		(*BALANCE*)
		(*************************************************************************************************)
		bI_EnableBalanceLink                                            := TRUE;
		fI_CorrectionValue                                              := 1.00;
		iI_RefreshRate                                                  := 2000;   (*ms*)
		FOR iL_Counter := 1 TO iCIk_NB_INKSTORAGE_TANK DO
			sAdsIkInkStorageTank[iL_Counter].sI_EnableBalance.bI_Command  := TRUE;

			sAdsIkInkStorageTank[iL_Counter].sI_InkDensitySet.fI_Val      := 1.07;
			sAdsIkInkStorageTank[iL_Counter].sI_CorrectionValue.fI_Val    := 1.00;
			sAdsIkInkStorageTank[iL_Counter].fO_StorageTankSize           := 25.0;   (*l*)

			sAdsIkInkStorageTank[iL_Counter].sI_WarningLevelSet.fI_Val    := 4.0;
			sAdsIkInkStorageTank[iL_Counter].sI_ErrorlevelSet.fI_Val      := 3.0;
			sAdsIkInkStorageTank[iL_Counter].sI_MaintenanceTimeout.lI_Val := 5000;

      (*Varnish parameter*)
      sAdsIkInkStorageTank[iL_Counter].sI_InkParameter.aWaveform           := 'waveform.wav';
      sAdsIkInkStorageTank[iL_Counter].sI_InkParameter.sTemperature.fI_Val := 35.0;
      sAdsIkInkStorageTank[iL_Counter].sI_InkParameter.sMeniscus.fI_Val    := -24.5;
      sAdsIkInkStorageTank[iL_Counter].sI_InkParameter.sDensity.fI_Val     := 1.0;
      sAdsIkInkStorageTank[iL_Counter].sI_InkParameter.sViscosity.fI_Val   := 100.0;
		END_FOR

		FOR iL_Counter := 1 TO iCIk_NB_INKBALANCE DO
      fL_BalanceOffset[iL_Counter]                                  := 0;

			sAdsIkInkStorageTank[iL_Counter].aI_CalibrateFrameText1       := 'aaaaaaaa';
			sAdsIkInkStorageTank[iL_Counter].aI_CalibrateFrameText2       := 'bbbbbbbb';
		END_FOR;
		sAdsIkInkStorageTank[1].aI_CalibrateFrameText1                  := '4D5A2406';
		sAdsIkInkStorageTank[1].aI_CalibrateFrameText2                  := '399128E6';
		sAdsIkInkStorageTank[2].aI_CalibrateFrameText1                  := '4D5426F9';
		sAdsIkInkStorageTank[2].aI_CalibrateFrameText2                  := '3991CD5A';
		sAdsIkInkStorageTank[3].aI_CalibrateFrameText1                  := 'aaaaaaaa';
		sAdsIkInkStorageTank[3].aI_CalibrateFrameText2                  := 'bbbbbbbb';

    (*Recipe: load and write*)
    IF pFbRecipeMngr <> 0 THEN
      pFbRecipeMngr^.mWriteRecipe('');
      PRG_MACHINE.bI_RecipeValuesLoadedInk := TRUE;
    END_IF

  ELSE

    sR_RemVar_I.aL_Pattern := sR_RemVar_I.aL_Pattern;  (*TODO remove dummy code*)

    (*DEGASSING*)
    (*************************************************************************************************)
    sAdsIkDgas[1].bI_Enable             := sR_RemVar_I.lR_DgasEnable;
    sAdsIkDgas[1].sI_PressSet.fI_Val    := (sR_RemVar_I.fR_DgasPressStpt * sC_Config_I.fL_DGAS1_CONV_ADS_TO_LCL);

    bIDp_EnableMainDgasValve            := sR_RemVar_I.lR_DgasEnableMainValve;
    sC_Config_I.lL_DGAS_TIME_ERROR      := sR_RemVar_I.lR_DgasTimeError;


    (*MENISCUS*)
    (*************************************************************************************************)
    FOR iL_Counter := 1 TO iCIk_NB_MENC DO
      sAdsIkMenc[iL_Counter].bI_Enable                         := sR_RemVar_I.lR_MencEnable   [iL_Counter];
      sAdsIkMenc[iL_Counter].sI_PressSet.fI_Val                := sR_RemVar_I.fR_MencPressStpt[iL_Counter];
    END_FOR;

    sC_Config_I.wL_MENC_TIME_ERROR                             := sR_RemVar_I.wR_MencTimeError;
    sC_Config_I.wL_SUB_MENC_TIME_ERROR                         := sR_RemVar_I.wR_SubMencTimeError;


    (*SUB MENISCUS*)
    (*************************************************************************************************)
    (*Sub meniscus starts behind the meniscus*)
    FOR iL_Counter := 1 TO iCIk_NB_SUB_MENC DO
      sAdsIkMenc[iCIk_NB_MENC + iL_Counter].bI_Enable          := sR_RemVar_I.lR_SubMencEnable        [iL_Counter];
      sAdsIkMenc[iCIk_NB_MENC + iL_Counter].sI_PressSet.fI_Val := sR_RemVar_I.fR_SubMencPressStpt     [iL_Counter];
    END_FOR;


    (*INK*)
    (*************************************************************************************************)
    (*varnish*)
    FOR iL_Counter := 1 TO iCIk_NB_HEADERTANK DO
      sAdsIkHeaderTank[iL_Counter].sI_StoragetankAssignment.lI_Val    := sR_RemVar_I.lR_StoragetankAssignment[iL_Counter];
      sAdsIkHeaderTank[iL_Counter].sO_ActStoragetankAssignment.lI_Val := sR_RemVar_I.lR_ActStoragetankAssignment[iL_Counter];
      
      sAdsIkHeaderTank[iL_Counter].bI_EnableFillInk       := sR_RemVar_I.bI_EnableFillInk[iL_Counter];
      sAdsIkHeaderTank[iL_Counter].bI_FillModeAuto        := sR_RemVar_I.bI_FillModeAuto[iL_Counter];
      sAdsIkHeaderTank[iL_Counter].bI_EnableUnFillInk     := sR_RemVar_I.bI_EnableUnFillInk[iL_Counter];
      sAdsIkHeaderTank[iL_Counter].bI_UnFillModeAuto      := sR_RemVar_I.bI_UnFillModeAuto[iL_Counter];

      sAdsIkInkPump[iL_Counter].sI_InkPumpSpeedSet.lI_Val := WORD_TO_DINT(sR_RemVar_I.wR_StptSpeedFillInkPumpVarnishPercent[iL_Counter]);

      fb_Headertank[iL_Counter].StateHeadertank           := sR_RemVar_I.eR_StateHeadertank[iL_Counter];
    END_FOR

		wIDp_MinSpeedFillInkPumpVarnish								:= sR_RemVar_I.wR_MinSpeedFillInkPumpVarnish;
		wIDp_MaxSpeedFillInkPumpVarnish								:= sR_RemVar_I.wR_MaxSpeedFillInkPumpVarnish;
		wIDP_AnalogMinDigitVarnish 										:= sR_RemVar_I.wR_AnalogMinDigitVarnish;
		wIDP_AnalogMaxDigitVarnish 										:= sR_RemVar_I.wR_AnalogMaxDigitVarnish;
		wIDp_PumpTimeOffDelayVarnish									:= sR_RemVar_I.wR_PumpTimeOffDelayVarnish;

    lL_TimeReturnFlow                             := sR_RemVar_I.lR_TimeReturnFlow;
    lL_TimeBlowOut                                := sR_RemVar_I.lR_TimeBlowOut;
    lL_TimeEmptyCleaner                           := sR_RemVar_I.lR_TimeEmptyCleaner;
    lL_TimeWarnExchange                           := sR_RemVar_I.lR_TimeWarnExchange;

    sC_Config_I.wC_INKPUMP_MAX_TIME               := sR_RemVar_I.wR_InkPumpMaxTime;
    sC_Config_I.wC_CLEANERPUMP_MAX_TIME           := sR_RemVar_I.wR_CleanerPumpMaxTime;

    
    (*TEMP*)
    (*************************************************************************************************)
    FOR iL_Counter :=1 TO iCIk_NB_TEMP_CONTR DO
      sAdsIkHeater[iL_Counter].bI_EnableHeater     := sR_RemVar_I.bI_EnableHeater  [iL_Counter];
      sAdsIkHeater[iL_Counter].sI_HeaterSet.fI_Val := sR_RemVar_I.sI_HeaterSetPoint[iL_Counter];
    END_FOR


    (*PURGE*)
    (*************************************************************************************************)
    FOR iL_Counter := 1 TO iCIk_NB_PURGE_CONTR DO
      sAdsIkPurgeController[iL_Counter].bI_Enable         := sR_RemVar_I.bR_PurgeControllerEnable[iL_Counter];
    END_FOR;

    FOR iL_Counter := 1 TO iCIk_NB_PURGE_GROUP DO
      sAdsIkPurgeGroup[iL_Counter].bI_EnablePurge         := sR_RemVar_I.bR_PurgeGroupEnable       [iL_Counter];
      sAdsIkPurgeGroup[iL_Counter].bI_EnableThroughNozzle := sR_RemVar_I.bR_PurgeGroupThroughNozzle[iL_Counter];
      sAdsIkPurgeGroup[iL_Counter].bI_EnableFlush         := sR_RemVar_I.bR_PurgeGroupFlush        [iL_Counter];
    END_FOR;


		(*BALANCE*)
		(*************************************************************************************************)
		bI_EnableBalanceLink    := sR_RemVar_I.bI_EnableBalanceLink;
		fI_CorrectionValue      := sR_RemVar_I.fI_CorrectionValue;
		iI_RefreshRate          := sR_RemVar_I.iI_RefreshRate;
		iI_MaintenanceTimeout   := sR_RemVar_I.iI_MaintenanceTimeout;

		FOR iL_Counter := 1 TO iCIk_NB_INKSTORAGE_TANK DO
			sAdsIkInkStorageTank[iL_Counter].bI_EnableStorageTank        := sR_RemVar_I.bI_EnableStorageTank[iL_Counter];
			sAdsIkInkStorageTank[iL_Counter].lO_InkColorId               := sR_RemVar_I.lO_InkColorId[iL_Counter];
			sAdsIkInkStorageTank[iL_Counter].fO_StorageTankSize          := sR_RemVar_I.fO_StorageTankSize[iL_Counter];
		END_FOR;

		FOR iL_Counter := 1 TO iCIk_NB_INKBALANCE DO
			sAdsIkInkStorageTank[iL_Counter].sI_EnableBalance.bI_Command := sR_RemVar_I.bI_EnableBalance[iL_Counter];
			sAdsIkInkStorageTank[iL_Counter].sI_InkDensitySet.fI_Val     := sR_RemVar_I.sI_InkDensitySet[iL_Counter];
			sAdsIkInkStorageTank[iL_Counter].sI_CorrectionValue.fI_Val   := sR_RemVar_I.sI_CorrectionValue[iL_Counter];
			sAdsIkInkStorageTank[iL_Counter].sI_WarningLevelSet.fI_Val   := sR_RemVar_I.sI_WarningLevelSet[iL_Counter];
			sAdsIkInkStorageTank[iL_Counter].sI_ErrorlevelSet.fI_Val     := sR_RemVar_I.sI_ErrorlevelSet[iL_Counter];

      (*Varnish parameter*)
      sAdsIkInkStorageTank[iL_Counter].sI_InkParameter.iScannerId          := sR_RemVar_I.lR_VarParamScannerId[iL_Counter];
      sAdsIkInkStorageTank[iL_Counter].sI_InkParameter.iIndex              := sR_RemVar_I.iR_VarParamIndex[iL_Counter];
      sAdsIkInkStorageTank[iL_Counter].sI_InkParameter.sTemperature.fI_Val := sR_RemVar_I.fR_VarParamTemp[iL_Counter];
      sAdsIkInkStorageTank[iL_Counter].sI_InkParameter.sMeniscus.fI_Val    := sR_RemVar_I.fR_VarParamMenc[iL_Counter];
      sAdsIkInkStorageTank[iL_Counter].sI_InkParameter.aWaveform           := sR_RemVar_I.aR_VarParamWaveform[iL_Counter];
      sAdsIkInkStorageTank[iL_Counter].sI_InkParameter.iTimer              := sR_RemVar_I.iR_VarParamTimer[iL_Counter];
      sAdsIkInkStorageTank[iL_Counter].sI_InkParameter.sDensity.fI_Val     := sR_RemVar_I.fR_VarParamDensity[iL_Counter];
      sAdsIkInkStorageTank[iL_Counter].sI_InkParameter.sViscosity.fI_Val   := sR_RemVar_I.fR_VarParamViscosity[iL_Counter];
      sAdsIkInkStorageTank[iL_Counter].sI_InkParameter.iColorId            := sR_RemVar_I.iR_VarParamColorId[iL_Counter];
      FOR iL_Counter2 := 1 TO 10 DO
        sAdsIkInkStorageTank[iL_Counter].sI_InkParameter.bCompatibility[iL_Counter2] := sR_RemVar_I.bR_VarParamCompatibility[iL_Counter, iL_Counter2];
      END_FOR;

			sAdsIkInkStorageTank[iL_Counter].aI_CalibrateFrameText1      := sR_RemVar_I.aI_CalibrateFrameText1[iL_Counter];
			sAdsIkInkStorageTank[iL_Counter].aI_CalibrateFrameText2      := sR_RemVar_I.aI_CalibrateFrameText2[iL_Counter];

      fL_BalanceOffset[iL_Counter] := sR_RemVar_I.fR_BalanceOffset[iL_Counter];
		END_FOR;

  END_IF


  bL_RemVar_Init := FALSE;



(*************************************************************************************************)
(********************************* WRITING REMANENT VARIABLES ************************************)
(*************************************************************************************************)
ELSE

(*GENERAL*)
(*************************************************************************************************)
  sR_RemVar_I.aL_Pattern := 16#ABCD;

(*DEGASSING*)
(*************************************************************************************************)
  sR_RemVar_I.lR_DgasEnable           := sAdsIkDgas[1].bI_Enable;
  sR_RemVar_I.fR_DgasPressStpt        := sAdsIkDgas[1].sI_PressSet.fI_Val;

  sR_RemVar_I.lR_DgasEnableMainValve  := bIDp_EnableMainDgasValve;
  sR_RemVar_I.lR_DgasTimeError        := sC_Config_I.lL_DGAS_TIME_ERROR;

(*MENISCUS*)
(*************************************************************************************************)
  FOR iL_Counter := 1 TO iCIk_NB_MENC DO
    sR_RemVar_I.fR_MencPressStpt[iL_Counter]      := sAdsIkMenc[iL_Counter].sI_PressSet.fI_Val;
    sR_RemVar_I.lR_MencEnable   [iL_Counter]      := sAdsIkMenc[iL_Counter].bI_Enable;
  END_FOR;

  sR_RemVar_I.wR_MencTimeError                    := sC_Config_I.wL_MENC_TIME_ERROR;
  sR_RemVar_I.wR_SubMencTimeError                 := sC_Config_I.wL_SUB_MENC_TIME_ERROR;

(*SUB MENISCUS*)
(*************************************************************************************************)
  (*Sub meniscus starts behind the meniscus*)
  FOR iL_Counter := 1 TO iCIk_NB_SUB_MENC DO
    sR_RemVar_I.fR_SubMencPressStpt     [iL_Counter] := sAdsIkMenc[iCIk_NB_MENC + iL_Counter].sI_PressSet.fI_Val;
    sR_RemVar_I.lR_SubMencEnable        [iL_Counter] := sAdsIkMenc[iCIk_NB_MENC + iL_Counter].bI_Enable;
  END_FOR;

(*PURGE - GLOBAL*)
(*************************************************************************************************)
  FOR iL_Counter := 1 TO iCIk_NB_PURGE_CONTR DO
    sR_RemVar_I.bR_PurgeControllerEnable  [iL_Counter] := sAdsIkPurgeController[iL_Counter].bI_Enable;
  END_FOR;

  FOR iL_Counter := 1 TO iCIk_NB_PURGE_GROUP DO
    sR_RemVar_I.bR_PurgeGroupEnable       [iL_Counter] := sAdsIkPurgeGroup[iL_Counter].bI_EnablePurge;
    sR_RemVar_I.bR_PurgeGroupThroughNozzle[iL_Counter] := sAdsIkPurgeGroup[iL_Counter].bI_EnableThroughNozzle;
    sR_RemVar_I.bR_PurgeGroupFlush        [iL_Counter] := sAdsIkPurgeGroup[iL_Counter].bI_EnableFlush;
  END_FOR;


(*INK*)
(*************************************************************************************************)
  (*varnish*)
  FOR iL_Counter:= 1 TO iCIk_NB_HEADERTANK DO
    sR_RemVar_I.lR_StoragetankAssignment   [iL_Counter]           := sAdsIkHeaderTank[iL_Counter].sI_StoragetankAssignment.lI_Val;
    sR_RemVar_I.lR_ActStoragetankAssignment[iL_Counter]           := sAdsIkHeaderTank[iL_Counter].sO_ActStoragetankAssignment.lI_Val;
      
    sR_RemVar_I.bI_EnableFillInk  [iL_Counter]                    := sAdsIkHeaderTank[iL_Counter].bI_EnableFillInk;
    sR_RemVar_I.bI_FillModeAuto   [iL_Counter]                    := sAdsIkHeaderTank[iL_Counter].bI_FillModeAuto;
    sR_RemVar_I.bI_EnableUnFillInk[iL_Counter]                    := sAdsIkHeaderTank[iL_Counter].bI_EnableUnFillInk;
    sR_RemVar_I.bI_UnFillModeAuto [iL_Counter]                    := sAdsIkHeaderTank[iL_Counter].bI_UnFillModeAuto;

    sR_RemVar_I.wR_StptSpeedFillInkPumpVarnishPercent[iL_Counter] := DINT_TO_WORD(sAdsIkInkPump[iL_Counter].sI_InkPumpSpeedSet.lI_Val);
    
    sR_RemVar_I.eR_StateHeadertank[iL_Counter]                    := fb_Headertank[iL_Counter].StateHeadertank;
  END_FOR

	sR_RemVar_I.wR_MinSpeedFillInkPumpVarnish 				:= wIDp_MinSpeedFillInkPumpVarnish;
	sR_RemVar_I.wR_MaxSpeedFillInkPumpVarnish					:= wIDp_MaxSpeedFillInkPumpVarnish;
	sR_RemVar_I.wR_AnalogMinDigitVarnish 							:= wIDP_AnalogMinDigitVarnish;
	sR_RemVar_I.wR_AnalogMaxDigitVarnish 							:= wIDP_AnalogMaxDigitVarnish;
	sR_RemVar_I.wR_PumpTimeOffDelayVarnish 						:= wIDp_PumpTimeOffDelayVarnish;

  sR_RemVar_I.lR_TimeReturnFlow                     := lL_TimeReturnFlow;
  sR_RemVar_I.lR_TimeBlowOut                        := lL_TimeBlowOut;
  sR_RemVar_I.lR_TimeEmptyCleaner                   := lL_TimeEmptyCleaner;
  sR_RemVar_I.lR_TimeWarnExchange                   := lL_TimeWarnExchange;

  sR_RemVar_I.wR_InkPumpMaxTime                     := sC_Config_I.wC_INKPUMP_MAX_TIME;
  sR_RemVar_I.wR_CleanerPumpMaxTime                 := sC_Config_I.wC_CLEANERPUMP_MAX_TIME;


(*RAMPE*)
(*************************************************************************************************)


(*TEMP*)
(*************************************************************************************************)
  FOR iL_Counter := 1 TO iCIk_NB_TEMP_CONTR DO
    sR_RemVar_I.bI_EnableHeater  [iL_Counter] := sAdsIkHeater[iL_Counter].bI_EnableHeater;
    sR_RemVar_I.sI_HeaterSetPoint[iL_Counter] := sAdsIkHeater[iL_Counter].sI_HeaterSet.fI_Val;
  END_FOR

  
(*INKSTORAGE_TANK*)
(*************************************************************************************************)
  FOR iL_Counter := 1 TO iCIk_NB_INKSTORAGE_TANK DO
    sR_RemVar_I.bI_EnableStorageTank[iL_Counter] := sAdsIkInkStorageTank[iL_Counter].bI_EnableStorageTank;
    sR_RemVar_I.lO_InkColorId[iL_Counter]        := sAdsIkInkStorageTank[iL_Counter].lO_InkColorId;
    sR_RemVar_I.fO_StorageTankSize[iL_Counter]   := sAdsIkInkStorageTank[iL_Counter].fO_StorageTankSize;
  END_FOR;

	(*BALANCE*)
	sR_RemVar_I.bI_EnableBalanceLink  := bI_EnableBalanceLink;
	sR_RemVar_I.fI_CorrectionValue    := fI_CorrectionValue;
	sR_RemVar_I.iI_RefreshRate        := iI_RefreshRate;
	sR_RemVar_I.iI_MaintenanceTimeout := iI_MaintenanceTimeout;

  FOR iL_Counter := 1 TO iCIk_NB_INKBALANCE DO
    sR_RemVar_I.bI_EnableBalance    [iL_Counter]   := sAdsIkInkStorageTank[iL_Counter].sI_EnableBalance.bI_Command;
    sR_RemVar_I.sI_InkDensitySet    [iL_Counter]   := sAdsIkInkStorageTank[iL_Counter].sI_InkDensitySet.fI_Val;
    sR_RemVar_I.sI_CorrectionValue  [iL_Counter]   := sAdsIkInkStorageTank[iL_Counter].sI_CorrectionValue.fI_Val;
    sR_RemVar_I.sI_WarningLevelSet  [iL_Counter]   := sAdsIkInkStorageTank[iL_Counter].sI_WarningLevelSet.fI_Val;
    sR_RemVar_I.sI_ErrorlevelSet    [iL_Counter]   := sAdsIkInkStorageTank[iL_Counter].sI_ErrorlevelSet.fI_Val;

    (*Varnish parameter*)
    sR_RemVar_I.lR_VarParamScannerId[iL_Counter]   := sAdsIkInkStorageTank[iL_Counter].sI_InkParameter.iScannerId;
    sR_RemVar_I.iR_VarParamIndex    [iL_Counter]   := sAdsIkInkStorageTank[iL_Counter].sI_InkParameter.iIndex;
    sR_RemVar_I.fR_VarParamTemp     [iL_Counter]   := sAdsIkInkStorageTank[iL_Counter].sI_InkParameter.sTemperature.fI_Val;
    sR_RemVar_I.fR_VarParamMenc     [iL_Counter]   := sAdsIkInkStorageTank[iL_Counter].sI_InkParameter.sMeniscus.fI_Val;
    sR_RemVar_I.aR_VarParamWaveform [iL_Counter]   := sAdsIkInkStorageTank[iL_Counter].sI_InkParameter.aWaveform;
    sR_RemVar_I.iR_VarParamTimer    [iL_Counter]   := sAdsIkInkStorageTank[iL_Counter].sI_InkParameter.iTimer;
    sR_RemVar_I.fR_VarParamDensity  [iL_Counter]   := sAdsIkInkStorageTank[iL_Counter].sI_InkParameter.sDensity.fI_Val;
    sR_RemVar_I.fR_VarParamViscosity[iL_Counter]   := sAdsIkInkStorageTank[iL_Counter].sI_InkParameter.sViscosity.fI_Val;
    sR_RemVar_I.iR_VarParamColorId  [iL_Counter]   := sAdsIkInkStorageTank[iL_Counter].sI_InkParameter.iColorId;
    FOR iL_Counter2 := 1 TO 10 DO
      sR_RemVar_I.bR_VarParamCompatibility[iL_Counter, iL_Counter2] := sAdsIkInkStorageTank[iL_Counter].sI_InkParameter.bCompatibility[iL_Counter2];
    END_FOR;

    sR_RemVar_I.aI_CalibrateFrameText1[iL_Counter] := sAdsIkInkStorageTank[iL_Counter].aI_CalibrateFrameText1;
    sR_RemVar_I.aI_CalibrateFrameText2[iL_Counter] := sAdsIkInkStorageTank[iL_Counter].aI_CalibrateFrameText2;

    sR_RemVar_I.fR_BalanceOffset[iL_Counter] := fL_BalanceOffset[iL_Counter];
  END_FOR;

END_IF;
END_ACTION

ACTION Simulate:
IF bL_SimInputs THEN
  
  FOR iL_CounterDgas := 1 TO iCIk_NB_DGAS DO
    fb_DgasMencContr[iL_CounterDgas].iI_ActValue := LREAL_TO_INT(fb_DgasMencContr[iL_CounterDgas].pSetValue * fb_DgasMencContr[iL_CounterDgas].fR_ConvAdsToLocal);
  
    sAdsIkDgas[iL_CounterDgas].bI_Enable := TRUE;
  END_FOR
  
  FOR iL_CounterMenc := 1 TO iCIk_NB_MENC_STA DO
    fb_MeniscusMencContr[iL_CounterMenc].iI_ActValue := LREAL_TO_INT(fb_MeniscusMencContr[iL_CounterMenc].pSetValue * fb_MeniscusMencContr[iL_CounterMenc].fR_ConvAdsToLocal);
  
    sAdsIkMenc[iL_CounterMenc].bI_Enable := TRUE;
  END_FOR
  
  bIKn_TankCleanerLevelEmpty := TRUE;
  bIKn_TankRefuseLevelFull   := TRUE;
  
  FOR iL_Counter := 1 TO iCIk_NB_TEMP_HYS DO
    fb_TempControllerHys[iL_Counter].iI_ActValue := DINT_TO_INT(fb_TempControllerHys[iL_Counter].pSetValue);
  END_FOR
END_IF

// init any storage tank assignement
FOR iL_Counter := 1 TO iCIk_NB_HEADERTANK DO
  IF sAdsIkHeaderTank[iL_Counter].sI_StoragetankAssignment.lI_Val = 0 THEN
    sAdsIkHeaderTank[iL_Counter].sI_StoragetankAssignment.lI_Val := UDINT_TO_DINT(sL_BLK_INKSTORAGE_TANK[1].iBlk_AdsId);
	END_IF
END_FOR
END_ACTION

ACTION Visu:
(*call visu controls*)
fb_VisuDgasMencController    (sI_Ary_Fb := fb_DgasMencContr    , sI_Ary_Ads := sAdsIkDgas);
fb_VisuMeniscusMencController(sI_Ary_Fb := fb_MeniscusMencContr, sI_Ary_Ads := sAdsIkMenc);
END_ACTION

END_PROGRAM

// ---- POUs/Products/Ink/FB_PurgeControllerSequence.TcPOU
FUNCTION_BLOCK FB_PurgeControllerSequence EXTENDS FB_PurgeController
VAR_INPUT
  iSubMencPos                  : I_AirVolume;
  iSubMencNeg                  : I_AirVolume;
END_VAR

VAR_OUTPUT
  bO_DeactivateLevelControlHT  : BOOL;
  bO_DeactivateSubMencNeg      : BOOL;

  bO_PurgeReleaseValveDelayed  AT %Q* : BOOL;              (*Purge pressure release valve*)
END_VAR

VAR
  _bActivateSequence           : BOOL;

  iL_PurgeStep                 : INT := 0;
  fb_TonSubMencRelease         : TON;
  fb_TonSubMencReleaseDelay    : TON;
  fb_TonSubMencReactivate      : TON;
  fb_RTrigCommand              : R_TRIG;
  fb_SubMencPosRamp            : FB_SPEED_RAMP;
  fb_SubMencNegRamp            : FB_SPEED_RAMP;
END_VAR

VAR PERSISTENT
  tR_ReleaseTime               : TIME := T#3S;
  tR_SubMencReleaseDelay       : TIME := T#1S;
  tR_SubMencReactivateTime     : TIME := T#2S;
  iR_SubMencPosFactor          : INT  := 50;
  iR_SubMencNegFactor          : INT  := 50;
  tR_SubMencPosRampTime        : INT  := 10;
  tR_SubMencNegRampTime        : INT  := 10;
END_VAR

VAR CONSTANT
  iC_StepIdle                  : INT := 0;
  iC_StepMencRelease           : INT := 1;
  iC_StepLevelContr            : INT := 2;
  iC_StepPurge                 : INT := 3;
  iC_StepReactivate1           : INT := 4;
  iC_StepReactivate2           : INT := 5;
END_VAR

(*Delay for one ReleaseValve*)
bO_PurgeReleaseValveDelayed := fbPurgeGroup[1].bO_PurgeReleaseValve;

IF _bActivateSequence THEN
  CASE iL_PurgeStep OF
    iC_StepIdle:  (*Idle, wait for start command*)
      IF     (   _pAdsIf^.sI_ActivatePurge.bI_Command
              OR IbPurgeContrRequestHT
              OR (iMachineInk.pPurgeRequest AND (   _pAdsIf^.sI_ActivatePurge.bO_CommandCanEx
                                                 OR bL_PurgeAuto)))
         AND _pAdsIf^.sI_ActivatePurge.bO_CommandCanEx
      THEN
        _pAdsIf^.sI_ActivatePurge.bO_CommandExec := TRUE;
        _pAdsIf^.sI_ActivatePurge.bI_Command     := FALSE;
  
        fb_TonSubMencRelease(IN := FALSE);
        FOR iL_CounterPurgeGroup := 1 TO iL_RegPurgeGroupItfs DO
          fb_TonSubMencReleaseDelay(IN := FALSE);
        END_FOR
        fb_RTrigCommand(CLK := _pAdsIf^.sI_ActivatePurge.bI_Command);
  
        fb_SubMencPosRamp(bI_EnableRamp := TRUE, bI_StartRamp := FALSE, II_SpeedActPercent := 100);
        fb_SubMencNegRamp(bI_EnableRamp := TRUE, bI_StartRamp := FALSE, II_SpeedActPercent := 100);
  
        iL_PurgeStep := iC_StepMencRelease;
      ELSE
        SUPER^();  
  
        bO_DeactivateLevelControlHT := FALSE;
        bO_DeactivateSubMencNeg     := FALSE;
      END_IF
  
    iC_StepMencRelease:  (*Release sub menc pressure*)
      fb_TonSubMencRelease(IN:= TRUE, PT := tR_ReleaseTime);
  
      FOR iL_CounterPurgeGroup := 1 TO iL_RegPurgeGroupItfs DO
        fb_TonSubMencReleaseDelay(IN := TRUE, PT := tR_SubMencReleaseDelay);
        bO_PurgeReleaseValveDelayed := fb_TonSubMencReleaseDelay.Q;
  
        fbPurgeGroup[iL_CounterPurgeGroup].pEnableValve := TRUE;
      END_FOR
      
      IF fb_TonSubMencRelease.Q THEN
        iL_PurgeStep := iC_StepLevelContr;
      END_IF
    
      (*Abort Purge*)
      fb_RTrigCommand(CLK := _pAdsIf^.sI_ActivatePurge.bI_Command);
      IF fb_RTrigCommand.Q THEN
        fb_TonSubMencReactivate(IN := FALSE);
  
        iL_PurgeStep := iC_StepReactivate1;
      END_IF
    
    iC_StepLevelContr:
      bO_DeactivateLevelControlHT := TRUE;
  
      _pAdsIf^.sI_ActivatePurge.bI_Command := TRUE;
    
      iL_PurgeStep := iC_StepPurge;
    
    iC_StepPurge:
      SUPER^();  
      IF _bBusy THEN
        _pAdsIf^.sI_ActivatePurge.bI_Command := FALSE;
      ELSE
        fb_TonSubMencReactivate(IN := FALSE);
  
        iL_PurgeStep := iC_StepReactivate1;
      END_IF
  
    iC_StepReactivate1:
      fb_TonSubMencReactivate(IN:= TRUE, PT := tR_SubMencReactivateTime);
  
      (*SubMenc must be run up by ramp*)
      fb_SubMencPosRamp( bI_StartRamp         := TRUE
                       , II_XTimeRamp         := tR_SubMencPosRampTime
                       , II_YAnalogMinPercent := iR_SubMencPosFactor
                       , II_YAnalogMaxPercent := 100);
      iSubMencPos.pPressSetFactor := DINT_TO_REAL(fb_SubMencPosRamp.IO_YPercent) / 100;
      
      bO_DeactivateLevelControlHT := FALSE;
      bO_DeactivateSubMencNeg     := TRUE;
  
      _pAdsIf^.sI_ActivatePurge.bO_CommandExec := FALSE;
      _pAdsIf^.sI_ActivatePurge.bI_Command     := FALSE;
  
      FOR iL_CounterPurgeGroup := 1 TO iL_RegPurgeGroupItfs DO
        fbPurgeGroup[iL_CounterPurgeGroup].pEnableValve := FALSE;
      END_FOR
  
      IF fb_TonSubMencReactivate.Q THEN
        iL_PurgeStep := iC_StepReactivate2;
      END_IF
    
    iC_StepReactivate2:
      (*SubMenc must be run up by ramp*)
      fb_SubMencPosRamp( bI_StartRamp         := TRUE
                       , II_XTimeRamp         := tR_SubMencPosRampTime
                       , II_YAnalogMinPercent := iR_SubMencPosFactor
                       , II_YAnalogMaxPercent := 100);
      iSubMencPos.pPressSetFactor := DINT_TO_REAL(fb_SubMencPosRamp.IO_YPercent) / 100;
      fb_SubMencNegRamp( bI_StartRamp         := TRUE
                       , II_XTimeRamp         := tR_SubMencNegRampTime
                       , II_YAnalogMinPercent := iR_SubMencNegFactor
                       , II_YAnalogMaxPercent := 100);
      iSubMencNeg.pPressSetFactor := DINT_TO_REAL(fb_SubMencNegRamp.IO_YPercent) / 100;
  
      bO_DeactivateSubMencNeg := FALSE;
  
      IF fb_SubMencPosRamp.bO_MaxSpeedReached AND fb_SubMencNegRamp.bO_MaxSpeedReached THEN
        iSubMencPos.pPressSetFactor := 1;
        iSubMencNeg.pPressSetFactor := 1;
        
        iL_PurgeStep := iC_StepIdle;
      END_IF
    
  END_CASE
ELSE
  SUPER^();  
END_IF

PROPERTY pActivateSequence : BOOL
SET
_bActivateSequence := pActivateSequence;
END_SET
END_PROPERTY

END_FUNCTION_BLOCK

// ---- POUs/Products/Ink/InkCirculation/FB_InkCirculation.TcPOU
FUNCTION_BLOCK FB_InkCirculation EXTENDS FB_BaseInk IMPLEMENTS I_SleepObserver, I_EmergencyObserver

VAR_INPUT
  InActValue                 AT %I* : INT;                      (*Actual value*)
  IbActValueWcState          AT %I* : BOOL;                     (*EM3701 pressure WcState*)
  IbInkLevelReachedBack      AT %I* : BOOL;                     (*HT back level reached*)

  iPurgeController                  : I_Purge;
  iMencController                   : I_AirVolume;

  IbEnable                          : BOOL;                     (*Enable function*)
  IbAxisMovement                    : BOOL;                     (*Axis movement*)
  IbHeadertankOk                    : BOOL;                     (*Headertank ok*)
  IbPHTempOk                        : BOOL;                     (*Printhead temperature ok*)
END_VAR

VAR_OUTPUT
  ObHtCloseInkConnectionValve       : BOOL;                     (*HT: close ink connection valve front to back*)
  ObHtCloseMencConnectionValve      : BOOL;                     (*HT back: close menc connection valve*)
  ObValveActivation                 : BOOL;                     (*HT: valve activation*)
  ObPumpActivation                  : BOOL;                     (*HT: pump activation*)
END_VAR

VAR
  _sName                            : STRING;                   (*Block name*)

  _bEStop                           : BOOL := FALSE;            (*EStop active*)
  _bSleep                           : BOOL := FALSE;            (*Sleep active*)
  bCheckParameterError01            : BOOL := FALSE;            (*CheckParameter: error 01 reported*)
  bLevelError                       : BOOL := FALSE;            (*HT back level error*)
  bCirculationActive                : BOOL;                     (*Circulation active*)
  bConditionsMet                    : BOOL;                     (*Conditions met*)
  bPumpActivation                   : BOOL;                     (*HT: pump activation*)
  fbTpPumpOn                        : TP;                       (*HT: pump activation on*)
  tPumpOnTime                       : TIME;                     (*HT: pump activation on*)
  fbTpPumpWait                      : TP;                       (*HT: pump activation wait*)
  tPumpWaitTime                     : TIME;                     (*HT: pump activation wait*)
  bResetErrorCounter                : BOOL;                     (*Reset HT back level error counter*)

  fbTonSubMencOK                    : TON;                      (*Sub menc pressure ok*)
  fbTonNoMovement                   : TON;                      (*No axis movement active*)
  fbTonResumeCirculation            : TON;                      (*Resume circulation after level error*)

  fSubMencActValue                  : LREAL;                    (*HT: actual pressure of back side*)
  fSubMencTargetValue               : LREAL;                    (*HT: target pressure of back side*)
END_VAR

VAR PERSISTENT
  tRSubMencOk                       : TIME := T#5S;             (*Supervision time for sub menc ok*)
  tRNoMovement                      : TIME := T#1M;             (*Supervision time axis movement*)
  tRResumeCirculation               : TIME := T#1M;             (*Resume circulation after level error*)
  tRPumpDutyCycleFrequency          : TIME := T#100MS;          (*Frequency for duty cycle of pump*)
  nRPumpDutyCycle                   : UINT := 30;               (*Duty cycle of pump*)

  fRConvAdsToLocal                  : LREAL := 10.0;            (*Factor to convert from ADS to local*)
  fRSubMencDeltaP                   : LREAL := -2.5;            (*HT: delta pressure of sub menc on back side*)
  fRSubMencHysteresisP              : LREAL :=  0.5;            (*HT: hysteresis pressure*)
  fRSubMencCorrectionP              : LREAL :=  0.0;            (*HT: correction pressure*)

  nRErrorCounter                    : UINT := 0;                (*HT back level error counter*)
END_VAR

(*--- check parameter -------------------*)
IF NOT mCheckParameter() THEN RETURN; END_IF

(*HT back error*)
IF bCirculationActive AND IbInkLevelReachedBack THEN
  bLevelError    := TRUE;
  nRErrorCounter := nRErrorCounter + 1;
END_IF
fbTonResumeCirculation(IN := bLevelError, PT := tRResumeCirculation);
IF fbTonResumeCirculation.Q THEN
  bLevelError    := FALSE;
END_IF
IF bResetErrorCounter THEN
  nRErrorCounter := 0;
END_IF

fbTonSubMencOK (IN := (iMencController.pErrorCode = 0), PT := tRSubMencOk);
fbTonNoMovement(IN := NOT IbAxisMovement, PT := tRNoMovement);

fSubMencActValue    := INT_TO_LREAL(InActValue) / fRConvAdsToLocal;
fSubMencActValue    := fSubMencActValue + fRSubMencCorrectionP;
fSubMencTargetValue := iMencController.pPressure + fRSubMencDeltaP;

bConditionsMet :=     NOT IbActValueWcState
                  AND NOT _bEStop
                  AND NOT _bSleep
                  AND NOT IbInkLevelReachedBack
                  AND NOT bLevelError
                  AND NOT iPurgeController.pPurgeBusy
                  AND fbTonSubMencOK.Q
                  AND fbTonNoMovement.Q
                  AND IbHeadertankOk
                  AND IbPHTempOk
                  AND (fRSubMencDeltaP <> 0);

IF IbEnable AND bConditionsMet THEN
  bCirculationActive           := TRUE;
  ObHtCloseInkConnectionValve  := TRUE;
  ObHtCloseMencConnectionValve := TRUE;
  ObValveActivation            := TRUE;

  IF fSubMencActValue >= (fSubMencTargetValue + fRSubMencHysteresisP) THEN
    bPumpActivation := TRUE;
  END_IF
  IF fSubMencActValue <= (fSubMencTargetValue - fRSubMencHysteresisP) THEN
    bPumpActivation := FALSE;
  END_IF
ELSE  
  bCirculationActive           := FALSE;
  ObHtCloseInkConnectionValve  := FALSE;
  ObHtCloseMencConnectionValve := FALSE;
  ObValveActivation            := FALSE;
  bPumpActivation              := FALSE;
END_IF

(*Pump is activated with a variable duty cycle*)
tPumpOnTime   := DINT_TO_TIME((TIME_TO_DINT(tRPumpDutyCycleFrequency) * nRPumpDutyCycle) / 100);
tPumpWaitTime := DINT_TO_TIME((TIME_TO_DINT(tRPumpDutyCycleFrequency) * (100 - nRPumpDutyCycle)) / 100);
IF bPumpActivation THEN
  IF (nRPumpDutyCycle = 0) THEN
    ObPumpActivation := FALSE;
  ELSIF (nRPumpDutyCycle = 100) THEN
    ObPumpActivation := TRUE;
  ELSE
    fbTpPumpOn  (IN := NOT fbTpPumpWait.Q, PT := tPumpOnTime);
    fbTpPumpWait(IN := NOT fbTpPumpOn.Q  , PT := tPumpWaitTime);
  
    ObPumpActivation := fbTpPumpOn.Q;
  END_IF
ELSE
  fbTpPumpOn  (IN := FALSE);
  fbTpPumpWait(IN := FALSE);

  ObPumpActivation := FALSE;
END_IF

(*
  Check if all necessary variables are properly defined 
  - check if initialized
  - crash prevention!
*)
METHOD PRIVATE mCheckParameter : BOOL
IF (iPurgeController = 0) OR (iMencController = 0) THEN
  IF NOT bCheckParameterError01 THEN
    bCheckParameterError01 := TRUE;
    F_Report_Error(Report_Error_0Pointer);
  END_IF
  RETURN;
END_IF

mCheckParameter := TRUE; // all params ok
END_METHOD

METHOD mEmergencyUpdate
VAR_INPUT
	(*updated estop value TRUE = active*)
	bEStop	: BOOL;
END_VAR
_bEStop := bEStop;
END_METHOD

METHOD mSleepUpdate
VAR_INPUT
	(*updated sleep value TRUE = active*)
	bSleep	: BOOL;
END_VAR
_bSleep := bSleep;
END_METHOD

PROPERTY pName : STRING
SET
_sName := pName;
END_SET
END_PROPERTY

END_FUNCTION_BLOCK

// ---- POUs/Projects/Machine/PRG_MACHINE.TcPOU
PROGRAM PRG_MACHINE
(*************************************************************************************************)
(*  FILENAME:    PRG_MACHINE.EXP                                                                 *)
(*  PROJECT:     CALMAR PUPLC                                                                    *)
(*  COPYRIGHT:   All rights reserved (c) Wifag//Polytype, Fribourg/Switzerland (2016)            *)
(*  ENVIRONMENT: TwinCAT PLC                                                                     *)
(*  VERSION:     <version>                                                                       *)
(*************************************************************************************************)
(*  DESCRIPTION:                                                                   <description> *)
(*    Controls the machine functionalities.                                                      *)
(*     - System command: sleep/wake up, emergency stop, air ok.                                  *)
(*    Messaging: - fb_Msg[1] := `eCMa_EMERGENCY_STOP_ACTIVE`                                     *)
(*               - fb_Msg[2] := `eCMa_MACHINE_DISABLED`                                          *)
(*               - fb_Msg[3] := `eCMa_MACHINE_COMM_ERR`                                          *)
(*               - fb_Msg[4] := `eCMa_SLEEP_MODE_ACTIVE`                                         *)
(*               - fb_Msg[5] := `eCMa_TEMPERATURE_MONITORING`                                    *)
(*               - fb_Msg[6] := `eCMa_STOR_TANKS_DISABLED`                                       *)
(*               - fb_Msg[7] := `eCMa_INK_WC_STATE_ERROR`                                        *)
(*               - fb_Msg[8] := `eCMa_PRINT_WC_STATE_ERROR`                                      *)
(*               - fb_Msg[9] := `eCMa_MACHINE_WC_STATE_ERROR`                                    *)
(*               - fb_Msg[10]:= `eCMa_TCPIP_COMM_ERROR`                                          *)
(*               - fb_Msg[11]:= `eCIk_CLEANER_CONTAINER_LEVEL_EMPTY`                             *)
(*               - fb_Msg[12]:= `eCIk_REFUSE_CONTAINER_LEVEL_FULL`                               *)
(*               - fb_Msg[13]:= `eCMa_AXIS_ERROR_X_PNEUMATIC`                                    *)
(*               - fb_Msg[14]:= `eCMa_WATCH_CIRCUIT_BREAKER`                                     *)
(*               - fb_Msg[15]:= `eCMa_WATCH_FUSE_PH1`                                            *)
(*               - fb_Msg[16]:= `eCMa_WATCH_FUSE_HEATER1`                                        *)
(*               - fb_Msg[17]:= `eCMa_WATCH_CABINET_TEMP`                                        *)
(*               - fb_Msg[18]:= `eCMa_WATCH_SEPARATOR_NIVEAU`                                    *)
(*               - fb_Msg[19]:= `eCMa_AXIS_SAFETY_ACCEPTANCE`                                    *)
(*               - fb_Msg[20]:= `eCMa_DRIFT_CONTR_ERROR`                                         *)
(*               - fb_Msg[21]:= `eCIk_CLEAN_START_MISSING`                                       *)
(*               - fb_Msg[22]:= `eCMa_RECIPE_LOADED`                                             *)
(*               - fb_Msg[23]:= `eCMa_AXIS_ERROR_Z_PNEUMATIC`                                    *)
(*               - fb_Msg[24]:= `eCMa_CLEANER_TANK_INFO`                                         *)
(*               - fb_Msg[25]:= `eCMa_MAX_SPEED_EXCEEDED`                                        *)
(*               - fb_Msg[26]:= `eCMa_IMAGE_DEPTH_INCORRECT`                                     *)
(*               - fb_Msg[27]:= `eCMa_EXHAUST_SYSTEM_WARNING`                                    *)
(*               - fb_Msg[28]:= `eCMa_EXHAUST_SYSTEM_ERROR`                                      *)
(*               - fb_Msg[29]:= `eCMa_EXHAUST_SYSTEM_MALFUNCTION`                                *)
(*               - fb_Msg[30]:= `eCMa_CLEANER_TANK_FILLING`                                      *)
(*               - fb_Msg[31]:= `eCMa_SEPARATOR_LEVEL_REACHED`                                   *)
(*                                                                                </description> *)
(*************************************************************************************************)

VAR_INPUT
  bIKp_CircuitBreakerM1_Ok          AT %I*  : BOOL;   (*monitoring input*)
  bIKp_CircuitBreakerM2_Ok          AT %I*  : BOOL;   (*monitoring input*)
  bIKp_PowerSupply1M1_Ok            AT %I*  : BOOL;   (*monitoring input*)
  bIKp_PowerSupply2M1_Ok            AT %I*  : BOOL;   (*monitoring input*)
  bIKp_PowerSupply3M1_Ok            AT %I*  : BOOL;   (*monitoring input*)
  bIKp_PowerSupply1M2_Ok            AT %I*  : BOOL;   (*monitoring input*)
  bIKp_PowerSupply2M2_Ok            AT %I*  : BOOL;   (*monitoring input*)
  bIKp_PowerSupply3M2_Ok            AT %I*  : BOOL;   (*monitoring input*)
  bIKp_SefetyRelayOk                AT %I*  : ARRAY[1..iCPr_NB_PM] OF BOOL;   (*monitoring input*)
  bIKp_SafetyCoverOK                AT %I*  : ARRAY[1..iCPr_NB_PM] OF BOOL;   (*monitoring input*)
  bIKp_SafetyDoorsOK                AT %I*  : ARRAY[1..iCPr_NB_PM] OF BOOL;   (*monitoring input*)

  bIKp_CabinetTemp_Ok               AT %I*  : BOOL;   (*monitoring input*)
  bIKp_SeparatorNiveau_Ok           AT %I*  : ARRAY[1..iCPr_NB_PM] OF BOOL;   (*-BX66: monitoring input*)
  
  (*Beckhoff EAP interface*)
  InEAP_WatchdogCycleIndex          AT %I*  : INT;    (*Watchdog: check CycleIndex*)
  InEAP_OperatingMode               AT %I*  : BYTE;   (*Operating mode*)
  IbEAP_ShutDownActive              AT %I*  : BOOL;   (*Master is shutting down*)                          (*not used yet*)
  IbEAP_Engaged                     AT %I*  : ARRAY[1..iCPr_NB_PM] OF BOOL;   (*DEM engaged*)
  IbEAP_PrintEnabled                AT %I*  : ARRAY[1..iCPr_NB_PM] OF BOOL;   (*Print enabled*)
  IbEAP_EStop                       AT %I*  : BOOL;   (*Emergency stop*)
  IbEAP_StandbyActive               AT %I*  : BOOL;   (*Standby active*)
  IbEAP_MessageReset                AT %I*  : BOOL;   (*Message reset*)       (*used in PRG_System*)
  IbEAP_PinningClosed               AT %I*  : ARRAY[1..iCPr_NB_PM] OF BOOL;   (*Pinning shutter closed*)
  IbEAP_CleaningStart               AT %I*  : ARRAY[1..iCPr_NB_PM] OF BOOL;   (*Start cleaning*)           (*not used yet*)
  InEAP_SubstrateThickness          AT %I*  : DINT;   (*Substrate thickness [µm]*)
  InEAP_SubstrateWidth              AT %I*  : DINT;   (*Substrate width [µm]*)                             (*not used yet*)
  InEAP_FormatLength                AT %I*  : DINT;   (*Format length [µm]*)
  InEAP_WebStretchFactor            AT %I*  : DINT;   (*Web stretch factor [0/00]*)
  InEAP_LateralRegister             AT %I*  : DINT;   (*Lateral register [µm]*)
  IbEAP_SpliceDetected              AT %I*  : ARRAY[1..iCPr_NB_PM] OF BOOL;   (*Splice detected*)
  InEAP_Module2ToModule3            AT %I*  : DINT;   (*Distance between Module 2 and 3 [µm]*)
  IbEAP_TargetSpeedReached          AT %I*  : BOOL;   (*Target speed reached*)
  InEAP_NeutralFibreFactor          AT %I*  : DINT;   (*Neutral fibre factor [%]*)
  IbEAP_PrintMarksExist             AT %I*  : ARRAY[1..iCPr_NB_PM] OF BOOL;   (*Print marks exist*)
  InEAP_TargetSpeed                 AT %I*  : DINT;   (*Neutral fibre factor [m/min]*)
  IbEAP_PanelLEDs                   AT %I*  : ARRAY[1..nC_MOTRONIC_PANEL_LEDS] OF BOOL;           (*Motronic panel LEDs*)

  (*Interfaces from other PRG*)
  fI_PrintingPosition                       : REAL;   (*Printing position [mm]*)
  bI_RecipeValuesLoadedInk                  : BOOL;
  bI_RecipeValuesLoadedPrint                : BOOL;
  bI_PrintActive                            : BOOL;   (*Printing active*)
  //bI_MachineStopped                         : BOOL;   (*Machine stopped*)
  sI_JobInkConsumption                      : ST_JOB_INK_CONSUMPTION; (*Job ink consumption information*)
  bI_PrintUnitStart                         : BOOL;   (*Printing unit start*)
  bI_PrintUnitStop                          : BOOL;   (*Printing unit stop*)
  lI_PrintedCopies                          : UDINT;  (*Printed copies*)
  bI_VacuumOk                               : BOOL;
  bI_CommandPrintlineExec                   : ARRAY[1..iCPr_NB_PM] OF BOOL;   (*Printline is executing*)

  (*Simulation*)
  bSimulation                               : BOOL;
END_VAR

VAR_OUTPUT
  bOKp_ResetFuse                    AT %Q*  : BOOL;   (*Reset WAGO Epsitron fuse*)
  ObPrinterReady                    AT %Q*  : BOOL;   (*Printer ready*)

  bO_SeparatorPumpDrainage          AT %Q*  : ARRAY[1..iCMa_NB_Cp] OF BOOL;   (* Enable separator pump for tank drainage (-MX196)*)

  bO_InitOk                                 : BOOL := FALSE;  (*Init Ok*)

  bO_WEUReady                               : ARRAY[1..iCPr_NB_PM] OF BOOL;  (*WEU ready*)

  (*Beckhoff EAP interface*)
  OnEAP_OperatingMode               AT %Q*  : BYTE;   (*Operating mode*)
  ObEAP_EngagingAllowed             AT %Q*  : ARRAY[1..iCPr_NB_PM] OF BOOL;   (*DEM engaging allowed*)
  ObEAP_EngagingActive              AT %Q*  : ARRAY[1..iCPr_NB_PM] OF BOOL;   (*DEM engaging active*)
  ObEAP_ShutdownReady               AT %Q*  : BOOL;   (*Shutdown ready*)
  ObEAP_StandbyReady                AT %Q*  : BOOL;   (*Standby ready*)
  ObEAP_PrintPosition               AT %Q*  : ARRAY[1..iCPr_NB_PM] OF BOOL;   (*Printing position*)
  ObEAP_MismatchLength              AT %Q*  : BOOL;   (*Mismatch length*)                               (*not used yet*)
  ObEAP_CleaningAllowed             AT %Q*  : ARRAY[1..iCPr_NB_PM] OF BOOL;   (*Cleaning allowed*)      (*not used yet*)
  ObEAP_CleaningActive              AT %Q*  : ARRAY[1..iCPr_NB_PM] OF BOOL;   (*Cleaning active*)
(*ToDo!!!*)   ObEAP_PrintReady                  AT %Q*  : ARRAY[1..iCPr_NB_PM] OF BOOL;   (*Ready to print*)
  OnEAP_VarnishQuantity             AT %Q*  : ARRAY[1..iCPr_NB_PM] OF DINT;   (*Varnish quantity [g/m^2]*)
  OnEAP_MaxWebSpeed                 AT %Q*  : DINT;   (*Max web speed [m/min]*)
  ObEAP_WarnungActive               AT %Q*  : BOOL;   (*Warning active*)
  ObEAP_ErrorActive                 AT %Q*  : BOOL;   (*Error active*)
  ObEAP_EStop                       AT %Q*  : BOOL;   (*Emergency stop / Fast stop*)
  OnEAP_PrintMarkPosBits            AT %Q*  : ARRAY[1..iCPr_NB_PM] OF WORD;   (*Print mark position (bit coded)*)
                                                                              (*Bit 0: no mark*)
                                                                              (*Bit 1: mark on drive side*)
                                                                              (*Bit 2: mark in center range*)
                                                                              (*Bit 3: mark on control side*)
  OnEAP_MasterSpeed                 AT %Q*  : ARRAY[1..iCPr_NB_PM] OF LREAL;  (*FB_POSITION_MASTER[x].fO_Master_Speed [m/s]*)
  ObPanelLEDs                       AT %Q*  : ARRAY[1..nC_MOTRONIC_PANEL_LEDS] OF BOOL;    (*Motronic panel LEDs*)

  (*Interfaces to other PRG*)
  bO_PrintUnitInPrintPosition               : ARRAY[1..iCPr_NB_PM] OF BOOL;    (*Print unit in print position*)
  bO_PrintUnitHigherWaitPosition            : ARRAY[1..iCPr_NB_PM] OF BOOL;    (*Print unit higher wait position*)
  bO_CleanPumpRequest                       : ARRAY[1..iCMa_NB_Cp] OF BOOL;    (* Request Cleaner Pump on*)
  sO_SystemCmd                              : ST_SYSTEM_CMD;
  bO_TotalWcState                           : BOOL := FALSE;   (*Monitoring: WcStates from all terminals*)
  bO_ErrorMsgActive                         : BOOL;   (*Error message at PUC active*)
  bO_WarningMsgActive                       : BOOL;   (*Warning message at PUC active*)
END_VAR

VAR
  iL_Counter                                : INT;    (*local iteration counter - default*)

  tskL_ActTaskInfo                          : PlcTaskSystemInfo;  (*CycleTime in multiple of 100ns*)
  Fb_GetCurTskIndx                          : GETCURTASKINDEX;
  lL_TaskCycleTime                          : REAL;  (*task cycle time [s]*)

  (* FB to store the generated block ID's *)
  bL_ExecuteBlockIdSave                     : BOOL;
  fb_BlkIdSave                              : FB_BLK_ID_SAVE;

  iL_Sel_BlkType                            : INT  := 1;          (*used for module information visualisation*)

  (*FAF: new cleaning station*)
  fB_Machine                                : FB_MachineState;
  
  fb_CleanProcess                           : ARRAY[1..iCMa_NB_Cp] OF FB_CleaningProcess;
  fb_CleaningCU                             : ARRAY[1..iCMa_NB_Cp] OF FB_CleaningMotorAxisCU;
  fb_CleaningCH                             : ARRAY[1..iCMa_NB_Cp] OF FB_CleaningMotorAxisCH;
  fb_CleaningPU                             : ARRAY[1..iCMa_NB_Cp] OF FB_CleaningMotorAxisPU;
  fb_CleaningValvePump                      : ARRAY[1..iCMa_NB_Cp] OF FB_Cleaning_ValvePump;
  fb_MotionInterlock                        : ARRAY[1..iCMa_NB_Cp] OF FB_MOTION_INTERLOCK;
  bL_RefKnownAll                            : BOOL;
  bL_AllInPosCappingClean                   : BOOL;

  (*Purge from machine*)
  fb_RFTrigPurgeBusy                        : ARRAY[1..iCMa_NB_Cp] OF RF_TRIG;
  fb_RFTrigCleanAfterPurge                  : ARRAY[1..iCMa_NB_Cp] OF RF_TRIG;
  fb_RTrigPurge                             : ARRAY[1..iCMa_NB_Cp] OF R_TRIG;
  fb_TonPurgeRequestTimeout                 : ARRAY[1..iCMa_NB_Cp] OF TON;

  fb_InterfaceMachineInk                    : ARRAY[1..iCPr_NB_PM] OF FB_IMachineInk;
  iMachineInk                               : ARRAY[1..iCPr_NB_PM] OF I_MachineInk;

  fb_MotionInkInterface                     : ARRAY[1..iCPr_NB_PM] OF FB_MOTION_TO_INKSYSTEM_IF;

  //fb_CU_EL7201                              : ARRAY[1..iCMa_NB_Cp] OF FB_EL7201_AXIS_CTRL;
  //fb_CH_EL7201                              : ARRAY[1..iCMa_NB_Cp] OF FB_EL7201_AXIS_CTRL;
  //fb_PU_EL7201                              : ARRAY[1..iCMa_NB_Cp] OF FB_EL7201_001_AXIS_CTRL;
  //lLCU_OffsetEncoder                        : ARRAY[1..iCMa_NB_Cp] OF DINT := [0,0];
  //lLCH_OffsetEncoder                        : ARRAY[1..iCMa_NB_Cp] OF DINT := [0,0];
  //lLPU_OffsetEncoder                        : ARRAY[1..iCMa_NB_Cp] OF DINT := [0,0];
  fb_RFTrigManualMoveCU                     : ARRAY[1..iCMa_NB_Cp] OF RF_TRIG;
  fb_RFTrigManualMoveCH                     : ARRAY[1..iCMa_NB_Cp] OF RF_TRIG;
  fb_RFTrigManualMovePU                     : ARRAY[1..iCMa_NB_Cp] OF RF_TRIG;
  sL_CU_CleanDevStatus                      : ARRAY[1..iCMa_NB_Cp] OF ST_CLEANING_DEV_STATUS;
  sL_CH_CleanDevStatus                      : ARRAY[1..iCMa_NB_Cp] OF ST_CLEANING_DEV_STATUS;
  sL_PU_CleanDevStatus                      : ARRAY[1..iCMa_NB_Cp] OF ST_CLEANING_DEV_STATUS;

  sADS_CleanProcess                         : ARRAY[1..iCMa_NB_Cp] OF ST_ADS_CLEAN_PROCESS;
  sADS_CleanAxis                            : ARRAY[1..iCMa_NB_Ca] OF ST_ADS_CLEAN_AXIS;
  sADS_Machine                              : ARRAY[1..iCMa_NB_Ma] OF ST_ADS_MACHINE;
  sC_Ads_Info                               : ST_ADS_INFO;
  sMappingInfo                              : T_MapInfo;        // Block mapping configuration
  ISystemBase                               : I_SystemBase;     // reference to system base
  pModuleDef                                : POINTER TO FB_ModuleDef;    // Module definition in system
  iSystemCmd                                : I_SystemCmd;                // System Command interface
  iSystemStatus                             : I_SystemStatus;             // System Status interface
  bAllowSleepFromMachine                    : BOOL;                       // enter sleep is allowed from machine
  rfTrig_Estop                              : RF_TRIG;
  
  
  bL_SafetyOk                               : ARRAY[1..iCPr_NB_PM] OF BOOL;
  bL_ResetAxis                              : BOOL;
  bL_MemMachineOn                           : BOOL := FALSE;

  (*Inputs from VISU*)
  (*
  nPrintModuleIdx                           : INT := 1;   (*PrintModule actual selection*)      
  fL_CuCappPurgPosition                     : REAL;  (*CU: capping/purge position [mm]*)
  fL_CuCleanRowPosition1                    : REAL;  (*CU: clean position 1 [mm]*)
  fL_CuCleanRowPosition2                    : REAL;  (*CU: clean position 2 [mm]*)
  fL_CuStopPosition                         : REAL;  (*CU: position ID for the lower limit [mm]*)
  fL_CuPlaceSpeed                           : REAL;  (*CU: speed for placement mouvement [mm/s]*)
  fL_CuWorkSpeed                            : REAL;  (*CU: speed for work mouvement [mm/s]*)
  fL_CuServiceSpeed                         : REAL;  (*CU: speed for maintenance operations [mm/s]*)
  fL_ChPositionP1                           : REAL;  (*CH: position P1 [mm]*)
  fL_ChPositionP2                           : REAL;  (*CH: position P2 [mm]*)
  fL_ChStopPosition                         : REAL;  (*CH: position ID for the lower limit [mm]*)
  fL_ChPlaceSpeed                           : REAL;  (*CH: speed for placement mouvement [mm/s]*)
  fL_ChWorkSpeed                            : REAL;  (*CH: speed for work mouvement [mm/s]*)
  fL_ChServiceSpeed                         : REAL;  (*CH: speed for maintenance operations [mm/s]*)
  fL_PuWaitingPosition                      : REAL;  (*PU: waiting position (Production Mode) [mm]*)
  fL_PuServicePosition                      : REAL;  (*PU: service position (Service Mode) [mm]*)
  fL_PuCleanPosition1                       : REAL;  (*PU: cleaning station moving position (Service Mode) [mm]*)
  fL_PuCleanPosition2                       : REAL;  (*PU: cleaning position (Service Mode) [mm]*)
  fL_PuStopPosition                         : REAL;  (*PU: position ID for the lower limit [mm]*)
  //fL_PuSetPositionValue                     : REAL;  (*PU: set position value [mm]*)
  fL_PuPlaceSpeed                           : REAL;  (*PU: speed for placement mouvement [mm/s]*)
  fL_PuWorkSpeed                            : REAL;  (*PU: speed for work mouvement [mm/s]*)
  fL_PuServiceSpeed                         : REAL;  (*PU: speed for maintenance operations [mm/s]*)
  wIDp_CleanerPumpLeadTime                  : WORD;  (*CH: lead time cleaner pump [ms]*)
  *)
  
  (*Initiation*)
  bL_RemVar_Init                            : BOOL;
  bL_DummyReadInput                         : BOOL;
  iL_DummyReadInput                         : INT;
  lL_DummyReadInput                         : DINT;

  fb_TonCheckMachineCom                     : TON;
  iL_MemWatchdogCycleIndex                  : INT;    (*Watchdog: check CycleIndex*)
  bL_WatchdogError                          : BOOL;

  (*Machine IOs*)
  bL_IO_MachineReady                        : BOOL;
  bL_IO_MachineHoming                       : BOOL;
  bL_IO_Engaged                             : ARRAY[1..iCPr_NB_PM] OF BOOL;
  //bL_IO_EStopOK                             : BOOL;
  bL_IO_StandbyActive                       : BOOL;
  bL_IO_PinningClosed                       : BOOL;
  lL_IO_SubstrateThickness                  : DINT;   (*Substrate thickness [µm]*)
  lL_IO_SubstrateWidth                      : DINT;   (*Substrate width [µm]*)
  lL_IO_FormatLength                        : DINT;   (*Format length [µm]*)
  fb_TonSeparatorLevel                      : ARRAY[1..iCMa_NB_Cp] OF TON;
  bL_SeparatorLevelReached                  : BOOL;

  bL_ProductionMode                         : ARRAY[1..iCPr_NB_PM] OF BOOL;   (*Production mode, not service mode*)

  bL_SleepVisu                              : BOOL;
  bL_WakeUpVisu                             : BOOL;
  fb_RTrigShutdownActive                    : R_TRIG;
  fb_FTrigShutdownActive                    : F_TRIG;
  fb_RTrigOpModeHoming                      : R_TRIG;
  fb_RTrigEngaged                           : ARRAY[1..iCPr_NB_PM] OF R_TRIG;
  fb_FTrigEngaged                           : ARRAY[1..iCPr_NB_PM] OF F_TRIG;
  fb_TonSleepToMachine                      : TON;

  fb_CappingCommandAfterEStop               : FB_CappingCommand;
  fb_CappingCommandAfterError               : ARRAY[1..iCPr_NB_PM] OF FB_CappingCommand;
  fb_CappingCommandAfterEngaged             : ARRAY[1..iCPr_NB_PM] OF FB_CappingCommand;
  fb_CappingCommandAfterShutdown            : ARRAY[1..iCPr_NB_PM] OF FB_CappingCommand;
  fb_CappingCommandAfterCleaning            : ARRAY[1..iCPr_NB_PM] OF FB_CappingCommand;
  _bCappingCommandAfterCleaning             : ARRAY[1..iCPr_NB_PM] OF BOOL;

  fb_TonAxisReady                           : ARRAY[1..iCPr_NB_PM] OF TON;
  fb_TonAxisReadyRelease                    : ARRAY[1..iCPr_NB_PM] OF TON;
  fb_RTrigCleaningFromMachine               : ARRAY[1..iCPr_NB_PM] OF R_TRIG;
  bL_CleaningCommandFromMachine             : ARRAY[1..iCPr_NB_PM] OF BOOL;
	fb_TofCleaningActive                      : ARRAY[1..iCPr_NB_PM] OF TOF;
  
  fb_TofPrintSystemOk                       : TOF;

  sC_Config_M                               : ST_CONFIG_M;

  (*Separator pump for tank drainage*)
  fb_TofSeparatorPumpNiveau                 : ARRAY[1..iCMa_NB_Cp] OF TOF;
  fb_TofSeparatorPumpPurge                  : ARRAY[1..iCMa_NB_Cp] OF TOF;

  bL_ManualVacuumBin                        : ARRAY[1..iCMa_NB_Cp] OF BOOL := [FALSE,FALSE];
  fb_RTrigManualVacuumBin                   : ARRAY[1..iCMa_NB_Cp] OF R_TRIG;
  fb_FTrigManualVacuumBin                   : ARRAY[1..iCMa_NB_Cp] OF F_TRIG;
  fb_RTrigPurgeVacuumBin                    : ARRAY[1..iCMa_NB_Cp] OF R_TRIG;
  fb_FTrigPurgeVacuumBin                    : ARRAY[1..iCMa_NB_Cp] OF F_TRIG;
  fb_FTrigSeparatorNiveau                   : ARRAY[1..iCMa_NB_Cp] OF F_TRIG;

  (*Compare sheet length with Image depth.*)
  lL_SubstrateLenPx                         : DINT;       (*Length of substrate [Px]*)
  lL_ImageDepthPx                           : DINT;       (*Image depth [Px]*)
  lL_ToleranceLenPx                         : DINT := 5;  (*Tolerance for compare sheet length with image depth [Px]*)
  bL_MismatchLength                         : BOOL;       (*Mismatch between length of substrate and image depth*)

  (*Messages*)
  fb_MsgQueueMachine                        : ARRAY [1..iCMa_NB_Ma] OF FB_MSG_QUEUE;
  fb_MachineMsgHandler                      : ARRAY [1..iCMa_NB_Ma] OF FB_MSG_HANDLER;
  sL_MsgConfigMachine                       : ARRAY [1..iCMa_NB_Ma] OF ST_MSG_CONFIG;
  fb_MachineMsg                             : ARRAY [1..iCMa_NB_Ma, 1..iCMa_NB_MSG] OF FB_MESSAGE;

  fb_TpResetFuse                            : TP;

  (*Machine communication NEW*)
  fbMachineComm                             : FB_MachineComm;
  
  (*Epsitron fuse control*)
  fbPowerControl                            : FB_WeuPowerControl;

  (*Exhaust system*)
  fb_ExhaustSystem                          :  ARRAY [1..iCPr_NB_PM] OF FB_ExhaustSystemPrint;
  

(* ADS Mappping *)
(*************************************************************************************************)
  iL_I                                      : INT;                (*instance counter*)
  iL_I2                                     : INT;                (*second instance counter for double loops*)
  sL_pI                                     : POINTER TO ST_MAP_BLK;  (*pointer to module mapping instance*)
  iL_Ctr                                    : INT;                (*counter value*)
  pL_Ctr                                    : POINTER TO INT;      (*pointer to mapping array index*)
  iL_ActElmt                                : INT;                (*actual array element*)
  aL_Name                                   : STRING;              (*Block string creation*)
  iL_NumModules                             : INT;                (*number of different block types*)
  cL_Module                                 : BYTE;                (*this module number*)

  FB_GEN_BLOCK_MAPPING                      : FB_GEN_BLOCK_MAPPING;   (*generation of block mappings in this module*)
  Fb_RegToAry                               : FB_REG_TO_ARY;      (**)

  sL_MOD_MAP                                : ARRAY [1..iCMa_NB_BLOCK_TYPES] OF ST_MAP_MODBLKARY;  (*array conataining all modules with their mapping informations*)
  sL_ModBlkAry                              : ST_MAP_MODBLKARY;

  sL_BLK_MA                                 : ARRAY [1..iCMa_NB_Ma] OF ST_MAP_BLK;      (*Machine*)
  sL_BLK_CP                                 : ARRAY [1..iCMa_NB_Cp] OF ST_MAP_BLK;      (*Cleaning process controller*)
  sL_BLK_AX                                 : ARRAY [1..iCMa_NB_Ca] OF ST_MAP_BLK;      (*array of all cleaning axes*)

  (*Recipe read/write*)
  pFbRecipeMngr                             : POINTER TO FB_RECIPE_READ_WRITE;
  bL_RecipeValuesLoadedMachine              : BOOL;

  (*Simulation variables*)
  bL_SimInputs                              : BOOL := FALSE;
END_VAR

VAR CONSTANT
(*GENERAL*)
(*************************************************************************************************)
  fC_TOLERANCE_PRINT_POSITION               : REAL := 0.001;       (*Tolerance for print position [m]*)

  cC_INIT                                   : BYTE := 16#00;      (*Operating mode: init*)
  cC_INITIALISED                            : BYTE := 16#00;      (*Operating mode: initialised*)
  cC_HOMING                                 : BYTE := 16#01;      (*Operating mode: homing*)
  cC_BASIC_HALT                             : BYTE := 16#02;      (*Operating mode: basic halt*)

  tC_DELAY_CAPPING_COMMAND                  : TIME := T#500MS;    (*Delay for automatic generated capping commands*)
  tC_RELEASE_CAPPING_COMMAND                : TIME := T#2S;       (*Release for automatic generated capping commands*)

  nC_MOTRONIC_PANEL_LEDS                    : INT  := 13;         (*Number Motronic panel LEDs*)
END_VAR

VAR PERSISTENT
  tR_TimeSeparatorPump                      : TIME := T#2M;   (*Separator pump for tank drainage*)
  tR_TimeSeparatorPump2                     : TIME := T#20S;  (*Separator pump for tank drainage*)

  tR_CleanerActivationAfterChange           : TIME := T#30S;
  lR_CleanerActivationAfterChange           : DINT := 30;          (*[%]*)
  bR_VaccumPumpActivationAfterCleanerChange : BOOL;

  tR_TimeSeparatorLevelCheck                : TIME := T#20S;   (*SeparatorLevel check*)
END_VAR

(* --------------------------------------------------------------------------------------------------------------- *)
(* Init                                                                                                            *)
(* --------------------------------------------------------------------------------------------------------------- *)
IF NOT bO_InitOk THEN
  Init();
  RETURN;
END_IF

(* --------------------------------------------------------------------------------------------------------------- *)
(* Execute module                                                                                                  *)
(* --------------------------------------------------------------------------------------------------------------- *)

(* Call ACTIONS *)
(*************************************************************************************************)
(*handle remanent variables*)
RemVar();

(*Epsitron fuse control*)
fbPowerControl();

(*Exhaust system*)
FOR iL_Counter := 1 TO iCPr_NB_PM DO
  fb_ExhaustSystem[iL_Counter](bI_PrintActive := bI_PrintActive);
END_FOR

(*Call simulation*)
Simulate();


(*-------------------------------------------------------------------------------------------------------------------*)
(* Infos from and to other tasks                                                                                     *)
(*-------------------------------------------------------------------------------------------------------------------*)
(*Ink infos are communicated via iMachineInk*)
bL_SeparatorLevelReached := FALSE;
FOR iL_Counter := 1 TO iCPr_NB_PM DO
  fb_TonSeparatorLevel[iL_Counter](IN := NOT bIKp_SeparatorNiveau_Ok[iL_Counter], PT := tR_TimeSeparatorLevelCheck);  (*ToDo*)
  bL_SeparatorLevelReached := bL_SeparatorLevelReached OR fb_TonSeparatorLevel[iL_Counter].Q;
  iMachineInk[iL_Counter]                    := fb_InterfaceMachineInk[iL_Counter];
  iMachineInk[iL_Counter].pSeparatorNiveauOk := NOT fb_TonSeparatorLevel[iL_Counter].Q;
  iMachineInk[iL_Counter].pInCappingPos      :=     fb_CleaningCU[iL_Counter].pInPosCappingClean
                                                AND (   fb_CleaningPU[iL_Counter].pInPosClean1
                                                     OR fb_CleaningPU[iL_Counter].pInPosClean2);
  iMachineInk[iL_Counter].pPurgeAllowed      :=     iMachineInk[iL_Counter].pSeparatorNiveauOk
                                                AND iMachineInk[iL_Counter].pInCappingPos;
  iMachineInk[iL_Counter].pEngaged           := bL_IO_Engaged[iL_Counter];
  iMachineInk[iL_Counter].pReceiptMessage    := fb_MsgQueueMachine[1].bO_ReceiptMessage;
END_FOR


fI_PrintingPosition      := PRG_PRINT.sAdsSheetAlignment[ePr_PU_UNIT_1].sI_HeadGap.fI_Val;
bI_PrintActive           := PRG_PRINT.FB_PU[ePr_PU_UNIT_1].sO_UnitStatus.bPrinting;
sI_JobInkConsumption     := PRG_PRINT.sAdsPrintUnit[ePr_PU_UNIT_1].sI_JobInkConsumption;
bI_PrintUnitStart        := PRG_PRINT.sAdsPrintUnit[ePr_PU_UNIT_1].sI_Start.bI_Command;
bI_PrintUnitStop         := PRG_PRINT.sAdsPrintUnit[ePr_PU_UNIT_1].sI_Stop.bI_Command;
lI_PrintedCopies         := PRG_PRINT.sAdsPrintUnit[ePr_PU_UNIT_1].lO_PrintedCopies;
bI_VacuumOk              := PRG_INK.bO_VacuumOk;

bO_ErrorMsgActive        := sADS_Machine[1].bI_ErrorMsgActive;
bO_WarningMsgActive      := sADS_Machine[1].bI_WarningMsgActive;

FOR iL_Counter := 1 TO iCPr_NB_PM DO
  bI_CommandPrintlineExec[iL_Counter] := PRG_INK.bO_CommandPrintlineExec[iL_Counter];
  bO_CleanPumpRequest    [iL_Counter] := fb_CleaningValvePump[iL_Counter].bO_CleanerPump;
END_FOR
    
(*-------------------------------------------------------------------------------------------------------------------*)
(*System command: sleep/wake up, emergency stop                                                                      *)
(*-------------------------------------------------------------------------------------------------------------------*)

(*EStop handling*)
iSystemCmd.setEmergencyState(bEmergency := IbEAP_EStop);
rfTrig_Estop(CLK:=IbEAP_EStop);

(*Sleep and WakeUp from machine*)
fb_RTrigShutdownActive(CLK := IbEAP_StandbyActive AND ObEAP_ShutdownReady);
fb_FTrigShutdownActive(CLK := IbEAP_StandbyActive);
IF fb_RTrigShutdownActive.Q THEN iSystemCmd.enterSleep('Machine'); END_IF
IF fb_FTrigShutdownActive.Q THEN iSystemCmd.exitSleep('Machine'); END_IF
IF bL_SleepVisu             THEN iSystemCmd.enterSleep('Visu'); bL_SleepVisu := FALSE; END_IF
IF bL_WakeUpVisu            THEN iSystemCmd.exitSleep('Visu'); bL_WakeUpVisu := FALSE; END_IF
IF fb_RTrigOpModeHoming.Q   THEN iSystemCmd.exitSleep('Homing'); END_IF 
bAllowSleepFromMachine := ObEAP_ShutdownReady;      // sleep canEx only if machine allows it

// setup intermediate variable still used everywhere
sO_SystemCmd.bEStop := iSystemStatus.bEmergency;
sO_SystemCmd.bSleep := iSystemStatus.bSleep;
sO_SystemCmd.bAirNotOk := FALSE;



FOR iL_Counter := 1 TO iCPr_NB_PM DO
  bL_SafetyOk[iL_Counter]        := NOT iSystemStatus.bEmergency           (*Safety ok for movement*)
                                    AND bIKp_SefetyRelayOk[iL_Counter]
                                    AND NOT bIKp_SafetyCoverOK[iL_Counter]
                                    AND NOT bIKp_SafetyDoorsOK[iL_Counter]
                                    AND (   IbEAP_PinningClosed[iL_Counter]
                                         OR bO_PrintUnitInPrintPosition[iL_Counter]
                                         OR (    fb_CleaningCU[iL_Counter].pInPosCappingClean
                                             AND fb_CleaningPU[iL_Counter].pInPosClean2));
END_FOR

sADS_Machine[1].bO_EmergencyStop := iSystemStatus.bEmergency;      (*Emergency stop*)
sADS_Machine[1].bO_MachineReady  := TRUE;                          (*Machine is switched on*)
sADS_Machine[1].bO_PrinterReady  := ObPrinterReady;

fB_Machine.bI_SafetyOk     := TRUE;
FOR iL_Counter := 1 TO iCPr_NB_PM DO
  fB_Machine.bI_SafetyOk   := fB_Machine.bI_SafetyOk AND bL_SafetyOk[iL_Counter];
END_FOR
fB_Machine.bI_MachineReady := NOT iSystemStatus.bEmergency AND (InEAP_OperatingMode >= cC_HOMING);


(*-------------------------------------------------------------------------------------------------------------------*)
(* Machine interface over Beckhoff EAP                                                                               *)
(*-------------------------------------------------------------------------------------------------------------------*)
(*Watchdog: check machine communication*)
fb_TonCheckMachineCom(IN := NOT fb_TonCheckMachineCom.Q, PT := T#1S);
IF fb_TonCheckMachineCom.Q THEN
  IF InEAP_WatchdogCycleIndex = iL_MemWatchdogCycleIndex THEN
    bL_WatchdogError := TRUE;
  ELSE
    bL_WatchdogError := FALSE;
  END_IF

  iL_MemWatchdogCycleIndex := InEAP_WatchdogCycleIndex;
END_IF

(*inputs*)
bL_IO_MachineReady               := (InEAP_OperatingMode >= cC_BASIC_HALT);
bL_IO_MachineHoming              := (InEAP_OperatingMode >= cC_HOMING);
fb_RTrigOpModeHoming(CLK := bL_IO_MachineHoming);

FOR iL_Counter := 1 TO iCPr_NB_PM DO
  (*Do prevent an abort of the axis if the engage will be toggled.*)
  fb_TonAxisReady[iL_Counter]( IN :=     sADS_CleanAxis[iCPr_MAP_Cp_CuAxis[iL_Counter]].bO_Ready
                                     AND sADS_CleanAxis[iCPr_MAP_Cp_ChAxis[iL_Counter]].bO_Ready
                                     AND sADS_CleanAxis[iCPr_MAP_Cp_PuAxis[iL_Counter]].bO_Ready
                             , PT := T#2S);
  (*Safety release: accept Engaged signal from Gallus if a ready signal misses for 30s.*)
  (*
  fb_TonAxisReadyRelease[iL_Counter]( IN := NOT (    sADS_CleanAxis[iCPr_MAP_Cp_CuAxis[iL_Counter]].bO_Ready
                                                 AND sADS_CleanAxis[iCPr_MAP_Cp_ChAxis[iL_Counter]].bO_Ready
                                                 AND sADS_CleanAxis[iCPr_MAP_Cp_PuAxis[iL_Counter]].bO_Ready)
                                    , PT := T#30S); *)
  IF fb_TonAxisReady[iL_Counter].Q (* OR fb_TonAxisReadyRelease[iL_Counter].Q *) THEN
    bL_IO_Engaged[iL_Counter] := IbEAP_Engaged[iL_Counter];
  END_IF
  // TEST
  IF IbEAP_PinningClosed[iL_Counter] THEN
    bL_IO_Engaged[iL_Counter] := IbEAP_Engaged[iL_Counter];
	END_IF
END_FOR


(*outputs*)
bL_RefKnownAll := TRUE;
FOR iL_Counter := 1 TO iCPr_NB_PM DO
  bL_RefKnownAll := bL_RefKnownAll AND fb_CleaningCU[iL_Counter].bL_RefKnown
                                   AND fb_CleaningCH[iL_Counter].bL_RefKnown
                                   AND fb_CleaningPU[iL_Counter].bL_RefKnown;
END_FOR

OnEAP_OperatingMode   := cC_INIT;         (*Operating mode*)
IF     NOT bL_RefKnownAll
   AND (InEAP_OperatingMode >= cC_HOMING)
THEN
  OnEAP_OperatingMode := cC_HOMING;       (*Operating mode*)
END_IF
IF bL_RefKnownAll THEN
  OnEAP_OperatingMode := cC_BASIC_HALT;   (*Operating mode*)
END_IF
FOR iL_Counter := 1 TO iCPr_NB_PM DO
  ObEAP_EngagingAllowed [iL_Counter] :=     NOT sO_SystemCmd.bSleep
                                        AND NOT iMachineInk[iL_Counter].pCleanExec
                                        AND NOT iMachineInk[iL_Counter].pPurgeBusy;
                                     (* AND NOT fb_Cleaning_Process.bO_MaintenanceActive*)
  ObEAP_EngagingActive  [iL_Counter] := IbEAP_Engaged[iL_Counter] AND NOT bO_PrintUnitHigherWaitPosition[iL_Counter];
  ObEAP_PrintPosition   [iL_Counter] := bO_PrintUnitInPrintPosition[iL_Counter];
  ObEAP_CleaningAllowed [iL_Counter] := ObEAP_ShutdownReady AND NOT fb_CleanProcess[iL_Counter].bI_CleanLocked;
  ObEAP_CleaningActive  [iL_Counter] := fb_TofCleaningActive[iL_Counter].Q;
  ObEAP_PrintReady      [iL_Counter] := bO_WEUReady[iL_Counter];
  OnEAP_VarnishQuantity [iL_Counter] := PRG_PRINT.sAdsPrintGroup[iCPr_MAP_PM_PG[iL_Counter]].sI_InkQuantity.lI_Val;
  IF IbEAP_PrintMarksExist[iL_Counter] THEN
    OnEAP_PrintMarkPosBits[iL_Counter] := fbMachineComm.sModuleMachineFeedback[iL_Counter].nPrintMarkPosBits;
  ELSE
    OnEAP_PrintMarkPosBits[iL_Counter] := 1; (*mark missing*) 
  END_IF
  OnEAP_MasterSpeed     [iL_Counter] := fbMachineComm.sModuleMachineFeedback[iL_Counter].fSpeed;
  (*TEST!!! use OnEAP_MasterSpeed to transmit PU position to Motronic*)
  OnEAP_MasterSpeed     [iL_Counter] := sADS_CleanAxis[iCPr_MAP_Cp_PuAxis[iL_Counter]].sO_AxisPosition.fO_Val;
END_FOR
(*Axis drive must be completed before the info 'ShutdownReady' goes to the machine.*)
bL_AllInPosCappingClean := TRUE;
FOR iL_Counter := 1 TO iCPr_NB_PM DO
  bL_AllInPosCappingClean := bL_AllInPosCappingClean AND fb_CleaningCU[iL_Counter].pInPosCappingClean AND fb_CleaningPU[iL_Counter].pInPosClean2;         (*Cleaning position*)
END_FOR
fb_TonSleepToMachine( IN := bL_AllInPosCappingClean         (*Cleaning position*)
                    , PT := T#1S);
ObEAP_ShutdownReady  := fb_TonSleepToMachine.Q;
ObEAP_StandbyReady   := sO_SystemCmd.bSleep AND ObEAP_ShutdownReady;
ObEAP_MismatchLength := bL_MismatchLength;
OnEAP_MaxWebSpeed    := fbMachineComm.nMaxSpeedMpMin;
ObEAP_WarnungActive  := sADS_Machine[1].bI_WarningMsgActive;
ObEAP_ErrorActive    := sADS_Machine[1].bI_ErrorMsgActive;
ObEAP_EStop := FALSE; 
FOR iL_Counter := 1 TO iCPr_NB_PM DO
  ObEAP_EStop := ObEAP_EStop OR bIKp_SafetyCoverOK[iL_Counter] OR bIKp_SafetyDoorsOK[iL_Counter];
END_FOR
FOR iL_Counter := 1 TO nC_MOTRONIC_PANEL_LEDS DO
  ObPanelLEDs[iL_Counter] := IbEAP_PanelLEDs[iL_Counter];
END_FOR

                       
(*-------------------------------------------------------------------------------------------------------------------*)
(* Check if image depth is different than format length                                                              *)
(*-------------------------------------------------------------------------------------------------------------------*)
lL_SubstrateLenPx := (F_MeterToSubPixel( fPosMeter  := DINT_TO_REAL(InEAP_FormatLength) * 0.000_001  (*[µm] => [m]*)
                                       , fResoSubPx := nC_PrintResolution * 1 (*Result should be in pixels*) ));
lL_ImageDepthPx   := (F_MeterToSubPixel( fPosMeter  := UDINT_TO_REAL(PRG_PRINT.sAdsPrintUnit[ePr_PU_UNIT_1].sI_JobSettings.lI_ImageDepth) * 0.000_001  (*[µm] => [m]*)
                                       , fResoSubPx := nC_PrintResolution * 1 (*Result should be in pixels*) ));
bL_MismatchLength :=    (lL_ImageDepthPx > (lL_SubstrateLenPx + lL_ToleranceLenPx))
                     OR (lL_ImageDepthPx < (lL_SubstrateLenPx - lL_ToleranceLenPx));
(*Reset error if*)
IF    PRG_PRINT.FB_PU[ePr_PU_UNIT_1].sO_PcFlags.bQueueEmpty                    (*no job loaded*)
   OR PRG_PRINT.sAdsPrintUnit[ePr_PU_UNIT_1].sI_JobSettings.lI_ImageDepth = 0  (*job setting invalid*)
   OR NOT PRG_PRINT.sAdsPrintUnit[ePr_PU_UNIT_1].bO_Ready                      (*job not started*)
   OR InEAP_FormatLength = 0                                                   (*0 length from machine*)
THEN
  bL_MismatchLength := FALSE;
END_IF


FOR iL_Counter := 1 TO iCPr_NB_PM DO
  (*Switch production / service mode*)
  fb_RTrigEngaged[iL_Counter](CLK := bL_IO_Engaged[iL_Counter]);
  IF fb_RTrigEngaged[iL_Counter].Q AND NOT iSystemStatus.bEmergency THEN
    bL_ProductionMode[iL_Counter] := TRUE;
  END_IF
  fb_FTrigEngaged[iL_Counter](CLK := bL_IO_Engaged[iL_Counter]);
  IF fb_FTrigEngaged[iL_Counter].Q THEN
    bL_ProductionMode[iL_Counter] := FALSE;
  END_IF
  IF     bL_IO_Engaged[iL_Counter]
     AND NOT iSystemStatus.bEmergency
     AND fbMachineComm.bMachineMoving
  THEN
    bL_ProductionMode[iL_Counter] := TRUE;
  END_IF
(*not needed here  
  IF NOT bL_IO_EStopOK THEN
    bL_ProductionMode[iL_Counter] := FALSE;
  END_IF
*)
END_FOR


IF NOT ObEAP_ShutdownReady THEN              (*Capping position*)
  (*Drive in capping after release of EStop*)
  fb_CappingCommandAfterEStop( IbTrigger := NOT iSystemStatus.bEmergency
                             , IbReset   := FALSE (*only internal reset*));

  FOR iL_Counter := 1 TO iCPr_NB_PM DO
    (*Drive in capping after release of axis error*)
    fb_CappingCommandAfterError   [iL_Counter]( IbTrigger :=     NOT sADS_CleanAxis[iCPr_MAP_Cp_CuAxis[iL_Counter]].bO_Error
                                                             AND NOT sADS_CleanAxis[iCPr_MAP_Cp_PuAxis[iL_Counter]].bO_Error
                                              , IbReset   := FALSE (*only internal reset*));
    (*Drive in capping after release of engaged*)
    fb_CappingCommandAfterEngaged [iL_Counter]( IbTrigger := NOT bL_IO_Engaged[iL_Counter]
                                              , IbReset   := bL_IO_Engaged[iL_Counter]);
    (*Drive in capping after shutdown received*)
    fb_CappingCommandAfterShutdown[iL_Counter]( IbTrigger := IbEAP_StandbyActive AND NOT bL_ProductionMode[iL_Counter]
                                              , IbReset   := NOT IbEAP_StandbyActive);
    (*Drive in capping after cleaning*)
    (*Not used, is done in state machine
    IF     (fb_CleanProcess[iL_Counter].sL_CurrentState^.sL_StateName = fb_CleanProcess[iL_Counter].fB_StateCleaning.pName)
       AND (fb_CleanProcess[iL_Counter].sL_CurrentState^.iL_State >= 3 (*cL_DONE*)) 
    THEN
      _bCappingCommandAfterCleaning[iL_Counter] := TRUE;
    END_IF
    fb_CappingCommandAfterCleaning[iL_Counter]( IbTrigger := _bCappingCommandAfterCleaning[iL_Counter]
                                              , IbReset   := FALSE (*only internal reset*));
    IF fb_CappingCommandAfterCleaning[iL_Counter].fb_TonReset.Q THEN 
      _bCappingCommandAfterCleaning[iL_Counter] := FALSE;
		END_IF
    *)
  END_FOR
END_IF


FOR iL_Counter := 1 TO iCPr_NB_PM DO
  (*Cleaning from Machine*)
  fb_RTrigCleaningFromMachine[iL_Counter](CLK := IbEAP_CleaningStart[iL_Counter]);
  IF fb_RTrigCleaningFromMachine[iL_Counter].Q THEN
    bL_CleaningCommandFromMachine[iL_Counter] := TRUE;
  END_IF
  IF fb_CleanProcess[iL_Counter].fB_StateCleaning.bL_DevOpActive OR NOT IbEAP_CleaningStart[iL_Counter] THEN
    bL_CleaningCommandFromMachine[iL_Counter] := FALSE;
  END_IF
END_FOR


(*-------------------------------------------------------------------------------------------------------------------*)
(* Interface to Substrate Transport PLC                                                                              *)
(*-------------------------------------------------------------------------------------------------------------------*)
ObPrinterReady :=     PRG_PRINT.bO_PrintSystemOk
                  AND PRG_INK.bO_InkSystemOk;

fb_TofPrintSystemOk(IN := PRG_PRINT.bO_PrintSystemOk, PT := T#10S); (*Delay for changing lay down amount without forcing basis machine to stop*)
FOR iL_Counter := 1 TO iCPr_NB_PM DO
  bO_WEUReady[iL_Counter] :=     PRG_PRINT.bO_PrintSystemOk  (*timer not needed here: fb_TofPrintSystemOk.Q*)
                             AND PRG_INK.bO_InkSystemOk
                             AND NOT fbMachineComm.sModuleMachineFeedback[iL_Counter].bSpeedExeeded
                             AND NOT bL_MismatchLength
             // not existing AND fb_ExhaustSystem[iL_Counter].bO_FUReady
                             AND NOT fb_ExhaustSystem[iL_Counter].bO_VacuumErrorLevel
                             AND NOT sO_SystemCmd.bSleep;
  // sim override
  IF bSimulation THEN 
    bO_WEUReady[iL_Counter] := TRUE;
  END_IF               
END_FOR


FOR iL_Counter := 1 TO iCMa_NB_Cp DO
  (*-------------------------------------------------------------------------------------------------------------------*)
  (* Motion Interlock                                                                                                   *)
  (*-------------------------------------------------------------------------------------------------------------------*)
  fb_MotionInterlock[iL_Counter].bIPU_PositionUnknown  := NOT fb_CleaningPU[iL_Counter].bL_RefKnown;
  fb_MotionInterlock[iL_Counter].bICU_PositionUnknown  := NOT fb_CleaningCU[iL_Counter].bL_RefKnown;
  fb_MotionInterlock[iL_Counter].fIPU_Position         := fb_CleaningPU[iL_Counter].fB_Axis.fO_ActualPosition;
  fb_MotionInterlock[iL_Counter].fICU_Position         := fB_CleaningCU[iL_Counter].fB_Axis.fO_ActualPosition;
  fb_MotionInterlock[iL_Counter].fCCU_CleaningPosition := fB_CleaningCU[iL_Counter].fI_PositionCappingClean / 1000;
  fb_MotionInterlock[iL_Counter].fCCU_SafePosition[2]  := fB_CleaningCU[iL_Counter].fI_PositionCappingClean / 1000;
  fb_MotionInterlock[iL_Counter].fCPU_SafePosition[1]  := fB_CleaningPU[iL_Counter].fI_PositionClean2 / 1000;
  fb_MotionInterlock[iL_Counter].fCPU_SafePosition[2]  := fB_CleaningPU[iL_Counter].fI_PositionClean1 / 1000;

  fb_MotionInterlock[iL_Counter]();

  
  (* --------------------------------------------------------------------------------------------------------------- *)
  (* Devices                                                                                                         *)
  (* --------------------------------------------------------------------------------------------------------------- *)
  fb_CleaningCU[iL_Counter]( bI_SafeToMove     := fb_MotionInterlock[iL_Counter].bOCU_MoveAuth);
  fb_CleaningCH[iL_Counter]( bI_SafeToMove     := fb_MotionInterlock[iL_Counter].bOCH_MoveAuth);
  fb_CleaningPU[iL_Counter]( bI_SafeToMove     := fb_MotionInterlock[iL_Counter].bOPU_MoveAuth
                           , fI_SheetThickness := DINT_TO_REAL(InEAP_SubstrateThickness) / 1000);
  fb_CleaningPU[iL_Counter].pPositionPrint := fI_PrintingPosition;

  IF sADS_CleanAxis[iCPr_MAP_Cp_CuAxis[iL_Counter]].bI_FaultAck OR bL_ResetAxis THEN fb_CleaningCU[iL_Counter].mAckError(); END_IF
  IF sADS_CleanAxis[iCPr_MAP_Cp_ChAxis[iL_Counter]].bI_FaultAck OR bL_ResetAxis THEN fb_CleaningCH[iL_Counter].mAckError(); END_IF
  IF sADS_CleanAxis[iCPr_MAP_Cp_PuAxis[iL_Counter]].bI_FaultAck OR bL_ResetAxis THEN fb_CleaningPU[iL_Counter].mAckError(); END_IF

  
  (*Manually empty cleaning tub*)
  fb_RTrigManualVacuumBin[iL_Counter](CLK := bL_ManualVacuumBin[iL_Counter]);
  fb_RTrigPurgeVacuumBin [iL_Counter](CLK := iMachineInk[iL_Counter].pPurgeBusy);
  IF     (   fb_RTrigManualVacuumBin[iL_Counter].Q
          OR fb_RTrigPurgeVacuumBin [iL_Counter].Q)
     AND bIKp_SeparatorNiveau_Ok[iL_Counter]
  THEN
    fb_CleaningValvePump[iL_Counter].pManuEmptyTub := TRUE;
  END_IF
  fb_FTrigManualVacuumBin[iL_Counter](CLK := bL_ManualVacuumBin[iL_Counter]);
  fb_FTrigPurgeVacuumBin [iL_Counter](CLK := iMachineInk[iL_Counter].pPurgeBusy);
  fb_FTrigSeparatorNiveau[iL_Counter](CLK := bIKp_SeparatorNiveau_Ok[iL_Counter]);
  IF     (   fb_FTrigManualVacuumBin[iL_Counter].Q 
          OR fb_FTrigPurgeVacuumBin [iL_Counter].Q
          OR fb_FTrigSeparatorNiveau[iL_Counter].Q)
     AND fb_CleaningValvePump[iL_Counter].pManuEmptyTub
  THEN
    fb_CleaningValvePump[iL_Counter].pManuEmptyTub := FALSE;
    bL_ManualVacuumBin[iL_Counter]                 := FALSE;
  END_IF


  (*Separator pump for tank drainage*)
  fb_TofSeparatorPumpNiveau[iL_Counter]( IN := NOT iSystemStatus.bEmergency AND NOT bIKp_SeparatorNiveau_Ok[iL_Counter]
                                       , PT := tR_TimeSeparatorPump);
  //while Purge (with off-delay)
  fb_TofSeparatorPumpPurge [iL_Counter]( IN := iMachineInk[iL_Counter].pPurgeBusy AND NOT PRG_INK.bO_TankRefuseLevelFull
                                       , PT := tR_TimeSeparatorPump2);
  bO_SeparatorPumpDrainage[iL_Counter] :=    fb_TofSeparatorPumpNiveau[iL_Counter].Q
                                          OR fb_TofSeparatorPumpPurge [iL_Counter].Q;

END_FOR


(* --------------------------------------------------------------------------------------------------------------- *)
(* Process                                                                                                         *)
(* --------------------------------------------------------------------------------------------------------------- *)
FOR iL_Counter := 1 TO iCMa_NB_Cp DO
  IF bL_ResetAxis THEN sADS_CleanProcess[iL_Counter].bI_AcknowledgeError := TRUE; END_IF

  fb_CleanProcess[iL_Counter].pI_ADS            := ADR(sADS_CleanProcess[iL_Counter]);
  fb_CleanProcess[iL_Counter].bI_UsrService     := NOT bL_ProductionMode[iL_Counter];
  fb_CleanProcess[iL_Counter].bI_UsrAbort       := iSystemStatus.bEmergency;
  (*HOA: not programmed yet!! fb_CleanProcess[iL_Counter].bI_MachineReady   := bL_IO_MachineReady AND bL_IO_EStop;*)
  fb_CleanProcess[iL_Counter].bI_CappingCommand :=    iMachineInk[iL_Counter].pCappingCommand
                                                   OR fb_CappingCommandAfterEStop.ObCappingCommand
                                                   OR fb_CappingCommandAfterError   [iL_Counter].ObCappingCommand
                                                   OR fb_CappingCommandAfterEngaged [iL_Counter].ObCappingCommand
                                                   OR fb_CappingCommandAfterShutdown[iL_Counter].ObCappingCommand
                                                   OR fb_CappingCommandAfterCleaning[iL_Counter].ObCappingCommand;
  fb_CleanProcess[iL_Counter].bI_PurgeCommand   := bL_CleaningCommandFromMachine[iL_Counter];
  fb_CleanProcess[iL_Counter].bI_CleanCommand   :=    iMachineInk[iL_Counter].pCleanCommand
                                                   OR fb_RFTrigCleanAfterPurge[iL_Counter].RT;
  fb_CleanProcess[iL_Counter].bI_CleanLocked    :=    NOT iMachineInk[iL_Counter].pSeparatorNiveauOk
                                                   OR iMachineInk[iL_Counter].pCleanerAirBubbleDetected;
  (*User settings from ADS*)
  fb_CleanProcess[iL_Counter].bI_UsrAutoMode        := sADS_CleanProcess[iL_Counter].bI_AutoMode;
  fb_CleanProcess[iL_Counter].bI_UsrCleanAfterCapp  := sADS_CleanProcess[iL_Counter].bI_CleanAfterCapp;  (*not used yet*)
  fb_CleanProcess[iL_Counter].bI_UsrCleanAfterPurge := sADS_CleanProcess[iL_Counter].bI_CleanAfterPurge OR bL_CleaningCommandFromMachine[iL_Counter];
  fb_CleanProcess[iL_Counter].bI_UsrPurgeAfterCapp  := sADS_CleanProcess[iL_Counter].bI_PurgeAfterCapp;  (*not used yet*)
  
  fb_CleanProcess[iL_Counter]();
  
  iMachineInk[iL_Counter].pCleanExec := fb_CleanProcess[iL_Counter].fB_StateCleaning.bL_DevOpActive;
  fb_TofCleaningActive[iL_Counter](IN := iMachineInk[iL_Counter].pCleanExec, PT := T#2S);

  (*Cleaning after Purge from CleanProcess if bI_UsrCleanAfterPurge is set.*)
  fb_RFTrigPurgeBusy      [iL_Counter](CLK := sADS_CleanProcess[iL_Counter].bO_PurgeExec AND iMachineInk[iL_Counter].pPurgeBusy);
  fb_RFTrigCleanAfterPurge[iL_Counter](CLK := fb_RFTrigPurgeBusy[iL_Counter].FT AND fb_CleanProcess[iL_Counter].bI_UsrCleanAfterPurge);
  
  (*Purge from machine*)
  fb_TonPurgeRequestTimeout[iL_Counter](IN := sADS_CleanProcess[iL_Counter].bO_PurgeExec, PT := T#30S);  (*Timeout if command can not executed.*)
  IF fb_TonPurgeRequestTimeout[iL_Counter].Q OR fb_RFTrigPurgeBusy[iL_Counter].FT THEN
    sADS_CleanProcess[iL_Counter].bO_PurgeExec := FALSE;
    iMachineInk[iL_Counter].pPurgeRequest      := FALSE;
  END_IF
  fb_RTrigPurge[iL_Counter](CLK := sADS_CleanProcess[iL_Counter].bO_PurgeExec AND fB_CleaningCU[iL_Counter].pInPosCappingClean);
  IF fb_RTrigPurge[iL_Counter].Q THEN
    iMachineInk[iL_Counter].pPurgeRequest := TRUE;
  END_IF
  
  (*Reset CanEx if VarnishChange is active*)
  IF bI_CommandPrintlineExec[iL_Counter] THEN
    sADS_CleanProcess[iL_Counter].bO_PurgeCanEx        := FALSE;
    sADS_CleanProcess[iL_Counter].bO_StartCappingCanEx := FALSE;
    sADS_CleanProcess[iL_Counter].bO_StopCappingCanEx  := FALSE;
    sADS_CleanProcess[iL_Counter].bO_CleanCanEx        := FALSE;
    sADS_CleanProcess[iL_Counter].bO_MaintenanceCanEx  := FALSE;
	END_IF
  (*Reset CanEx if separator niveau is reached*)
  IF NOT iMachineInk[iL_Counter].pSeparatorNiveauOk THEN
    sADS_CleanProcess[iL_Counter].bO_PurgeCanEx        := FALSE;
	END_IF
END_FOR


(*-------------------------------------------------------------------------------------------------------------------*)
(* Motion -> InkSystem Interface                                                                                     *)
(*-------------------------------------------------------------------------------------------------------------------*)
FOR iL_Counter := 1 TO iCMa_NB_Cp DO
  //fb_MotionInkInterface.sI_CleanDevCmd := fb_Cleaning_Process.sO_CleanDevCmd[4];
  fb_MotionInkInterface[iL_Counter].bI_CleanPumpOn := iMachineInk[iL_Counter].pCleanPumpRequest;
  fb_MotionInkInterface[iL_Counter].bI_PurgeBusy   := iMachineInk[iL_Counter].pPurgeBusy;
  
  fb_MotionInkInterface[iL_Counter]();
  
  iMachineInk[iL_Counter].pCleanPumpEnable := fb_MotionInkInterface[iL_Counter].bO_EnableCleanerPump;

  sADS_CleanAxis[iCPr_MAP_Cp_InkInterface[iL_Counter]].bO_Busy  := fb_MotionInkInterface[iL_Counter].sO_CleanDevStatus.bBusy;
  sADS_CleanAxis[iCPr_MAP_Cp_InkInterface[iL_Counter]].bO_Ready := fb_MotionInkInterface[iL_Counter].sO_CleanDevStatus.bReady;
  sADS_CleanAxis[iCPr_MAP_Cp_InkInterface[iL_Counter]].bO_Error := FALSE;
END_FOR


(*-------------------------------------------------------------------------------------------------------------------*)
(* Axes control                                                                                                      *)
(*-------------------------------------------------------------------------------------------------------------------*)
FOR iL_Counter := 1 TO iCMa_NB_Cp DO
  (*-------------------------------------------------------------------------------------------------------------------*)
  (* CLEAN UNIT MOTION CONTROL                                                                                         *)
  (*-------------------------------------------------------------------------------------------------------------------*)
  (*Manuell move in hand mode (NOT bI_UsrAutoMode)*)
  fb_RFTrigManualMoveCU[iL_Counter](CLK := sADS_CleanAxis[iCPr_MAP_Cp_CuAxis[iL_Counter]].bI_ManualMove);
  IF     NOT fb_CleanProcess[iL_Counter].bI_UsrAutoMode 
     AND fb_CleanProcess[iL_Counter].bI_UsrService
     AND bL_SafetyOk[iL_Counter]
  THEN
    sADS_CleanAxis[iCPr_MAP_Cp_CuAxis[iL_Counter]].bO_ManualMoveCanEx := TRUE;
  
    IF sADS_CleanAxis[iCPr_MAP_Cp_CuAxis[iL_Counter]].bI_ManualMove OR fb_RFTrigManualMoveCU[iL_Counter].FT THEN
      fB_CleaningCU[iL_Counter].mManuellMove( bI_Do                  := sADS_CleanAxis[iCPr_MAP_Cp_CuAxis[iL_Counter]].bI_ManualMove
                                            , fI_TargetPosition      := SEL( sADS_CleanAxis[iCPr_MAP_Cp_CuAxis[iL_Counter]].bI_ManualMove
                                                                           , (fb_CleaningCU[iL_Counter].fB_Axis.fO_ActualPosition * 1000)
                                                                           , sADS_CleanAxis[iCPr_MAP_Cp_CuAxis[iL_Counter]].fI_ManualTargetPos)
                                            , fL_ManualMoveTolerance := fb_CleaningCU[iL_Counter].fB_Axis.fI_Tolerance);
    END_IF
  ELSE
    sADS_CleanAxis[iCPr_MAP_Cp_CuAxis[iL_Counter]].bO_ManualMoveCanEx := FALSE;
    sADS_CleanAxis[iCPr_MAP_Cp_CuAxis[iL_Counter]].bI_ManualMove      := FALSE;
  
    IF fb_RFTrigManualMoveCU[iL_Counter].FT THEN
      fB_CleaningCU[iL_Counter].mManuellMove( bI_Do                  := FALSE
                                            , fI_TargetPosition      := (fb_CleaningCU[iL_Counter].fB_Axis.fO_ActualPosition * 1000)
                                            , fL_ManualMoveTolerance := fb_CleaningCU[iL_Counter].fB_Axis.fI_Tolerance);
    END_IF
  END_IF
  (*Rest command if move is done*)
  IF fB_CleaningCU[iL_Counter].bL_Ready OR fB_CleaningCU[iL_Counter].bL_Error THEN
    sADS_CleanAxis[iCPr_MAP_Cp_CuAxis[iL_Counter]].bI_ManualMove := FALSE;
	END_IF
  
  sL_CU_CleanDevStatus[iL_Counter] := fB_CleaningCU[iL_Counter].sStatus;
  
  (*ADS Feedback*)
  sADS_CleanAxis[iCPr_MAP_Cp_CuAxis[iL_Counter]].sO_AxisPosition.fO_Val := fB_CleaningCU[iL_Counter].fB_Axis.fO_ActualPosition * 1000;
  sADS_CleanAxis[iCPr_MAP_Cp_CuAxis[iL_Counter]].bO_Busy                := sL_CU_CleanDevStatus[iL_Counter].bBusy;
  sADS_CleanAxis[iCPr_MAP_Cp_CuAxis[iL_Counter]].bO_Ready               := sL_CU_CleanDevStatus[iL_Counter].bReady;
  sADS_CleanAxis[iCPr_MAP_Cp_CuAxis[iL_Counter]].wO_ErrorCode           := fB_CleaningCU[iL_Counter].wL_ErrorCode;
  sADS_CleanAxis[iCPr_MAP_Cp_CuAxis[iL_Counter]].bO_Error               := sL_CU_CleanDevStatus[iL_Counter].bError;

  
  (*-------------------------------------------------------------------------------------------------------------------*)
  (* CLEAN HEAD MOTION CONTROL                                                                                         *)
  (*-------------------------------------------------------------------------------------------------------------------*)
  (*Manuell move in hand mode (NOT bI_UsrAutoMode)*)
  fb_RFTrigManualMoveCH[iL_Counter](CLK := sADS_CleanAxis[iCPr_MAP_Cp_ChAxis[iL_Counter]].bI_ManualMove);
  IF     NOT fb_CleanProcess[iL_Counter].bI_UsrAutoMode 
     AND fb_CleanProcess[iL_Counter].bI_UsrService
     AND bL_SafetyOk[iL_Counter]
     AND fb_CleaningCU[iL_Counter].pInPosCappingClean
  THEN
    sADS_CleanAxis[iCPr_MAP_Cp_ChAxis[iL_Counter]].bO_ManualMoveCanEx := TRUE;
  
    IF sADS_CleanAxis[iCPr_MAP_Cp_ChAxis[iL_Counter]].bI_ManualMove OR fb_RFTrigManualMoveCH[iL_Counter].FT THEN
      fB_CleaningCH[iL_Counter].mManuellMove( bI_Do                  := sADS_CleanAxis[iCPr_MAP_Cp_ChAxis[iL_Counter]].bI_ManualMove
                                            , fI_TargetPosition      := SEL( sADS_CleanAxis[iCPr_MAP_Cp_ChAxis[iL_Counter]].bI_ManualMove
                                                                           , (fb_CleaningCH[iL_Counter].fB_Axis.fO_ActualPosition * 1000)
                                                                           , sADS_CleanAxis[iCPr_MAP_Cp_ChAxis[iL_Counter]].fI_ManualTargetPos)
                                            , fL_ManualMoveTolerance := fb_CleaningCH[iL_Counter].fB_Axis.fI_Tolerance);
    END_IF
  ELSE
    sADS_CleanAxis[iCPr_MAP_Cp_ChAxis[iL_Counter]].bO_ManualMoveCanEx := FALSE;
    sADS_CleanAxis[iCPr_MAP_Cp_ChAxis[iL_Counter]].bI_ManualMove      := FALSE;
  
    IF fb_RFTrigManualMoveCH[iL_Counter].FT THEN
      fB_CleaningCH[iL_Counter].mManuellMove( bI_Do                  := FALSE
                                            , fI_TargetPosition      := (fb_CleaningCH[iL_Counter].fB_Axis.fO_ActualPosition * 1000)
                                            , fL_ManualMoveTolerance := fb_CleaningCH[iL_Counter].fB_Axis.fI_Tolerance);
    END_IF
  END_IF
  (*Rest command if move is done*)
  IF fB_CleaningCH[iL_Counter].bL_Ready OR fB_CleaningCH[iL_Counter].bL_Error THEN
    sADS_CleanAxis[iCPr_MAP_Cp_ChAxis[iL_Counter]].bI_ManualMove := FALSE;
	END_IF

  sL_CH_CleanDevStatus[iL_Counter] := fB_CleaningCH[iL_Counter].sStatus;
  
  (*ADS Feedback*)
  sADS_CleanAxis[iCPr_MAP_Cp_ChAxis[iL_Counter]].sO_AxisPosition.fO_Val := fB_CleaningCH[iL_Counter].fB_Axis.fO_ActualPosition * 1000;
  sADS_CleanAxis[iCPr_MAP_Cp_ChAxis[iL_Counter]].bO_Busy                := sL_CH_CleanDevStatus[iL_Counter].bBusy;
  sADS_CleanAxis[iCPr_MAP_Cp_ChAxis[iL_Counter]].bO_Ready               := sL_CH_CleanDevStatus[iL_Counter].bReady;
  sADS_CleanAxis[iCPr_MAP_Cp_ChAxis[iL_Counter]].wO_ErrorCode           := fB_CleaningCH[iL_Counter].wL_ErrorCode;
  sADS_CleanAxis[iCPr_MAP_Cp_ChAxis[iL_Counter]].bO_Error               := sL_CH_CleanDevStatus[iL_Counter].bError;


  (*-------------------------------------------------------------------------------------------------------------------*)
  (* PRINT UNIT MOTION CONTROL                                                                                         *)
  (*-------------------------------------------------------------------------------------------------------------------*)
  (*Manuell move in hand mode (NOT bI_UsrAutoMode)*)
  fb_RFTrigManualMovePU[iL_Counter](CLK := sADS_CleanAxis[iCPr_MAP_Cp_PuAxis[iL_Counter]].bI_ManualMove);
  IF     NOT fb_CleanProcess[iL_Counter].bI_UsrAutoMode
     AND fb_CleanProcess[iL_Counter].bI_UsrService
     AND bL_SafetyOk[iL_Counter]
  THEN
    sADS_CleanAxis[iCPr_MAP_Cp_PuAxis[iL_Counter]].bO_ManualMoveCanEx := TRUE;
  
    IF sADS_CleanAxis[iCPr_MAP_Cp_PuAxis[iL_Counter]].bI_ManualMove OR fb_RFTrigManualMovePU[iL_Counter].FT THEN
      fb_CleaningPU[iL_Counter].mManuellMove( bI_Do                  := sADS_CleanAxis[iCPr_MAP_Cp_PuAxis[iL_Counter]].bI_ManualMove
                                            , fI_TargetPosition      := SEL( sADS_CleanAxis[iCPr_MAP_Cp_PuAxis[iL_Counter]].bI_ManualMove
                                                                           , (fb_CleaningPU[iL_Counter].fB_Axis.fO_ActualPosition * 1000)
                                                                           , sADS_CleanAxis[iCPr_MAP_Cp_PuAxis[iL_Counter]].fI_ManualTargetPos)
                                            , fL_ManualMoveTolerance := fb_CleaningPU[iL_Counter].fB_Axis.fI_Tolerance);
    END_IF
  ELSE
    sADS_CleanAxis[iCPr_MAP_Cp_PuAxis[iL_Counter]].bO_ManualMoveCanEx := FALSE;
    sADS_CleanAxis[iCPr_MAP_Cp_PuAxis[iL_Counter]].bI_ManualMove      := FALSE;
  
    IF fb_RFTrigManualMovePU[iL_Counter].FT THEN
      fb_CleaningPU[iL_Counter].mManuellMove( bI_Do                  := FALSE
                                            , fI_TargetPosition      := (fb_CleaningPU[iL_Counter].fB_Axis.fO_ActualPosition * 1000)
                                            , fL_ManualMoveTolerance := fb_CleaningPU[iL_Counter].fB_Axis.fI_Tolerance);
    END_IF
  END_IF
  (*Rest command if move is done*)
  IF fb_CleaningPU[iL_Counter].bL_Ready OR fb_CleaningPU[iL_Counter].bL_Error THEN
    sADS_CleanAxis[iCPr_MAP_Cp_PuAxis[iL_Counter]].bI_ManualMove := FALSE;
	END_IF

  (*Move to print position in production*)
  IF     bL_ProductionMode[iL_Counter]
     AND bL_IO_Engaged[iL_Counter]
     AND bL_SafetyOk[iL_Counter]
     AND fb_CleanProcess[iL_Counter].bI_UsrAutoMode
  THEN
    fb_CleaningPU[iL_Counter].mPrintPos( bI_PrintEnabled  := IbEAP_PrintEnabled[iL_Counter]
                                       , bI_PrintFinsihed := TRUE  (*ToDo: if PrintEnable is disabled, the print is to be finished first: b_PrintFinished[iL_Counter] OR IbEAP_SpliceDetected[iL_Counter]*)  );
  END_IF
  
  sL_PU_CleanDevStatus[iL_Counter] := fb_CleaningPU[iL_Counter].sStatus;
  
  (*ADS Feedback*)
  sADS_CleanAxis[iCPr_MAP_Cp_PuAxis[iL_Counter]].sO_AxisPosition.fO_Val := fb_CleaningPU[iL_Counter].fB_Axis.fO_ActualPosition * 1000;
  sADS_CleanAxis[iCPr_MAP_Cp_PuAxis[iL_Counter]].bO_Busy                := sL_PU_CleanDevStatus[iL_Counter].bBusy;
  sADS_CleanAxis[iCPr_MAP_Cp_PuAxis[iL_Counter]].bO_Ready               := sL_PU_CleanDevStatus[iL_Counter].bReady;
  sADS_CleanAxis[iCPr_MAP_Cp_PuAxis[iL_Counter]].wO_ErrorCode           := fb_CleaningPU[iL_Counter].wL_ErrorCode;
  sADS_CleanAxis[iCPr_MAP_Cp_PuAxis[iL_Counter]].bO_Error               := sL_PU_CleanDevStatus[iL_Counter].bError;

  (*Check if print unit is in print position*)
  bO_PrintUnitInPrintPosition   [iL_Counter] := fb_CleaningPU[iL_Counter].pInPosPrint;
  (*Check if print unit is higher than wait position*)
  bO_PrintUnitHigherWaitPosition[iL_Counter] := fb_CleaningPU[iL_Counter].pHigherPosWait;
END_FOR


(*-------------------------------------------------------------------------------------------------------------------*)
(* Handle new machine communication *)
fbMachineComm();


(*Fault Reset Generation*)
bL_ResetAxis    :=  rfTrig_Estop.FT OR ((InEAP_OperatingMode >= cC_HOMING) AND NOT bL_MemMachineOn); 
bL_MemMachineOn := (InEAP_OperatingMode >= cC_HOMING);


(*Machine messages*)
fb_MachineMsgHandler[1]();  (*Call to check for blocked access*)

fb_MachineMsg[1, 1](bI_Status := sADS_Machine[1].bO_EmergencyStop);
fb_MachineMsg[1, 2](bI_Status := NOT sADS_Machine[1].bO_MachineReady);
fb_MachineMsg[1, 3](bI_Event  := bL_WatchdogError);
fb_MachineMsg[1, 4](bI_Status := sO_SystemCmd.bSleep);
fb_MachineMsg[1, 5](bI_Status := NOT PRG_INK.bO_TemperatureOk OR NOT PRG_PRINT.bO_TemperatureOk);
fb_MachineMsg[1, 6](bI_Status := NOT PRG_INK.bO_InkStorageTankOk);
fb_MachineMsg[1, 7](bI_Status := PRG_INK.bO_TotalWcState);
fb_MachineMsg[1, 8](bI_Status := PRG_PRINT.bO_TotalWcState);
fb_MachineMsg[1, 9](bI_Status := bO_TotalWcState);
fb_MachineMsg[1,10](bI_Status := FALSE);
fb_MachineMsg[1,11](bI_Status := PRG_INK.bO_TankCleanerLevelEmpty);
fb_MachineMsg[1,12](bI_Status := PRG_INK.bO_TankRefuseLevelFull);
fb_MachineMsg[1,13](bI_Status := FALSE);
fb_MachineMsg[1,14](bI_Status :=    NOT bIKp_CircuitBreakerM1_Ok
                                 OR NOT bIKp_CircuitBreakerM2_Ok
                                 OR NOT bIKp_PowerSupply1M1_Ok
                                 OR NOT bIKp_PowerSupply2M1_Ok
                                 OR NOT bIKp_PowerSupply3M1_Ok
                                 OR NOT bIKp_PowerSupply1M2_Ok
                                 OR NOT bIKp_PowerSupply2M2_Ok
                                 OR NOT bIKp_PowerSupply3M2_Ok);
fb_MachineMsg[1,15](bI_Status := FALSE);
fb_MachineMsg[1,16](bI_Status := FALSE);
fb_MachineMsg[1,17](bI_Status := FALSE);    //NOT bIKp_CabinetTemp_Ok);
fb_MachineMsg[1,18](bI_Status := FALSE);
fb_MachineMsg[1,19](bI_Status := FALSE);
fb_MachineMsg[1,20](bI_Status := FALSE);
fb_MachineMsg[1,21](bI_Status := FALSE);  (*bO_CleanAborted*)
fb_MachineMsg[1,22](bI_Status := bL_RecipeValuesLoadedMachine OR bI_RecipeValuesLoadedInk OR bI_RecipeValuesLoadedPrint);
fb_MachineMsg[1,23](bI_Status := FALSE);
fb_MachineMsg[1,24](bI_Status := FALSE);
fb_MachineMsg[1,25](bI_Status := fbMachineComm.bSpeedExeeded);
fb_MachineMsg[1,26](bI_Status := bL_MismatchLength);
fb_MachineMsg[1,27](bI_Status := FALSE);
fb_MachineMsg[1,28](bI_Status := FALSE);
fb_MachineMsg[1,29](bI_Status := FALSE);
fb_MachineMsg[1,30](bI_Status := FALSE);
fb_MachineMsg[1,31](bI_Status := bL_SeparatorLevelReached);

fb_MsgQueueMachine[1]();

(*Reset fuses with message from GUI.*)
fb_TpResetFuse(IN := fb_MsgQueueMachine[1].bO_ReceiptMessage, PT := T#1S);
bOKp_ResetFuse := fb_TpResetFuse.Q;

IF fb_MsgQueueMachine[1].bO_ReceiptMessage THEN
  bL_RecipeValuesLoadedMachine := FALSE;
  bI_RecipeValuesLoadedInk     := FALSE;
  bI_RecipeValuesLoadedPrint   := FALSE;

  FOR iL_Counter := 1 TO iCPr_NB_PM DO
    iMachineInk[iL_Counter].pCleanerAirBubbleDetected := FALSE;

    fb_ExhaustSystem[iL_Counter].mAckError();
  END_FOR
  
  fbPowerControl.ackError();
END_IF


(*WcState: 0 = Data valid, 1 = Data invalid*)
bO_TotalWcState := FALSE;

(********************************* END OF PRG ****************************************************)

METHOD Init : BOOL
(* -- System & Module setup ---------------------------------------------------------------------*)
ISystemBase := PRG_SYSTEMBASE.getSystemBaseInterface();
IF ISystemBase = 0 THEN RETURN; END_IF
// Wait until system(base) is booted
IF ISystemBase.bBooting THEN RETURN; END_IF

